LIN {X -0.057,Y -490.852,Z 943.531,A 0.000,B 0.000,C 90.000,E1 275.511} C_DIS
LIN {X 0.167,Y -491.276,Z 943.528,A 0.000,B 0.000,C 90.000,E1 274.992} C_DIS
LIN {X -0.096,Y -491.294,Z 943.525,A 0.000,B 0.000,C 90.000,E1 274.531} C_DIS
LIN {X 0.132,Y -490.916,Z 943.522,A 0.000,B 0.000,C 90.000,E1 274.012} C_DIS
LIN {X -0.165,Y -489.960,Z 943.520,A 0.000,B 0.000,C 90.000,E1 273.555} C_DIS
LIN {X 0.056,Y -488.500,Z 943.517,A 0.000,B 0.000,C 90.000,E1 273.037} C_DIS
LIN {X -0.241,Y -486.374,Z 943.514,A 0.000,B 0.000,C 90.000,E1 272.579} C_DIS
LIN {X -0.058,Y -483.567,Z 943.511,A 0.000,B 0.000,C 90.000,E1 272.064} C_DIS
LIN {X 0.120,Y -479.943,Z 943.509,A 0.000,B 0.000,C 90.000,E1 271.547} C_DIS
LIN {X -0.213,Y -475.367,Z 943.506,A 0.000,B 0.000,C 90.000,E1 271.088} C_DIS
LIN {X -0.087,Y -469.751,Z 943.503,A 0.000,B 0.000,C 90.000,E1 270.573} C_DIS
LIN {X 0.011,Y -463.745,Z 943.501,A 0.000,B 0.000,C 90.000,E1 270.115} C_DIS
LIN {X 0.069,Y -457.400,Z 943.498,A 0.000,B 0.000,C 90.000,E1 269.714} C_DIS
LIN {X 0.079,Y -450.722,Z 943.497,A 0.000,B 0.000,C 90.000,E1 269.370} C_DIS
LIN {X 0.041,Y -443.908,Z 943.495,A 0.000,B 0.000,C 90.000,E1 269.083} C_DIS
LIN {X -0.122,Y -436.692,Z 943.494,A 0.000,B 0.000,C 90.000,E1 268.854} C_DIS
LIN {X 0.080,Y -429.536,Z 943.492,A 0.000,B 0.000,C 90.000,E1 268.625} C_DIS
LIN {X 0.075,Y -421.449,Z 943.491,A 0.000,B 0.000,C 90.000,E1 268.453} C_DIS
LIN {X -0.026,Y -412.042,Z 943.491,A 0.000,B 0.000,C 90.000,E1 268.339} C_DIS
LIN {X 0.076,Y -404.135,Z 943.491,A 0.000,B 0.000,C 90.000,E1 268.282} C_DIS
LIN {X 0.000,Y -181.172,Z 943.490,A 0.000,B 0.000,C 90.000,E1 268.282} C_DIS
LIN {X -0.046,Y -180.830,Z 943.472,A 0.000,B 0.000,C 90.000,E1 264.894} C_DIS
LIN {X 0.034,Y -178.935,Z 943.443,A 0.000,B 0.000,C 90.000,E1 259.803} C_DIS
LIN {X -0.099,Y -175.985,Z 943.415,A 0.000,B 0.000,C 90.000,E1 254.755} C_DIS
LIN {X 0.016,Y -175.481,Z 943.410,A 0.000,B 0.000,C 90.000,E1 253.866} C_DIS
LIN {X 0.072,Y -172.226,Z 943.387,A 0.000,B 0.000,C 90.000,E1 249.571} C_DIS
LIN {X 0.050,Y -171.704,Z 943.382,A 0.000,B 0.000,C 90.000,E1 248.720} C_DIS
LIN {X -0.025,Y -167.298,Z 943.353,A 0.000,B 0.000,C 90.000,E1 243.563} C_DIS
LIN {X -0.019,Y -166.677,Z 943.348,A 0.000,B 0.000,C 90.000,E1 242.692} C_DIS
LIN {X -0.028,Y -162.659,Z 943.324,A 0.000,B 0.000,C 90.000,E1 238.329} C_DIS
LIN {X 0.035,Y -161.348,Z 943.314,A 0.000,B 0.000,C 90.000,E1 236.548} C_DIS
LIN {X 0.077,Y -157.342,Z 943.290,A 0.000,B 0.000,C 90.000,E1 232.110} C_DIS
LIN {X 0.009,Y -155.328,Z 943.275,A 0.000,B 0.000,C 90.000,E1 229.461} C_DIS
LIN {X -0.060,Y -151.679,Z 943.250,A 0.000,B 0.000,C 90.000,E1 225.000} C_DIS
LIN {X -0.012,Y -150.543,Z 943.240,A 0.000,B 0.000,C 90.000,E1 223.176} C_DIS
LIN {X 0.021,Y -147.269,Z 943.215,A 0.000,B 0.000,C 90.000,E1 218.624} C_DIS
LIN {X -0.006,Y -145.297,Z 943.194,A 0.000,B 0.000,C 90.000,E1 214.978} C_DIS
LIN {X -0.014,Y -142.392,Z 943.164,A 0.000,B 0.000,C 90.000,E1 209.461} C_DIS
LIN {X 0.032,Y -141.372,Z 943.148,A 0.000,B 0.000,C 90.000,E1 206.668} C_DIS
LIN {X 0.010,Y -139.346,Z 943.112,A 0.000,B 0.000,C 90.000,E1 200.174} C_DIS
LIN {X 0.015,Y -139.019,Z 943.102,A 0.000,B 0.000,C 90.000,E1 198.308} C_DIS
LIN {X 0.011,Y -138.343,Z 943.055,A 0.000,B 0.000,C 90.000,E1 189.905} C_DIS
LIN {X 0.031,Y -139.392,Z 943.008,A 0.000,B 0.000,C 90.000,E1 181.489} C_DIS
LIN {X -0.056,Y -141.291,Z 942.972,A 0.000,B 0.000,C 90.000,E1 175.008} C_DIS
LIN {X 0.043,Y -142.654,Z 942.957,A 0.000,B 0.000,C 90.000,E1 172.186} C_DIS
LIN {X -0.007,Y -144.994,Z 942.931,A 0.000,B 0.000,C 90.000,E1 167.589} C_DIS
LIN {X -0.018,Y -147.621,Z 942.911,A 0.000,B 0.000,C 90.000,E1 163.921} C_DIS
LIN {X 0.061,Y -150.247,Z 942.890,A 0.000,B 0.000,C 90.000,E1 160.242} C_DIS
LIN {X -0.066,Y -153.642,Z 942.870,A 0.000,B 0.000,C 90.000,E1 156.666} C_DIS
LIN {X -0.008,Y -157.058,Z 942.850,A 0.000,B 0.000,C 90.000,E1 153.050} C_DIS
LIN {X 0.072,Y -161.188,Z 942.830,A 0.000,B 0.000,C 90.000,E1 149.459} C_DIS
LIN {X 0.020,Y -163.281,Z 942.821,A 0.000,B 0.000,C 90.000,E1 147.709} C_DIS
LIN {X 0.031,Y -167.724,Z 942.801,A 0.000,B 0.000,C 90.000,E1 144.196} C_DIS
LIN {X -0.057,Y -171.543,Z 942.787,A 0.000,B 0.000,C 90.000,E1 141.618} C_DIS
LIN {X -0.014,Y -176.485,Z 942.768,A 0.000,B 0.000,C 90.000,E1 138.162} C_DIS
LIN {X -0.016,Y -180.782,Z 942.753,A 0.000,B 0.000,C 90.000,E1 135.607} C_DIS
LIN {X -0.028,Y -186.189,Z 942.735,A 0.000,B 0.000,C 90.000,E1 132.243} C_DIS
LIN {X 0.037,Y -190.827,Z 942.721,A 0.000,B 0.000,C 90.000,E1 129.725} C_DIS
LIN {X 0.005,Y -194.361,Z 942.709,A 0.000,B 0.000,C 90.000,E1 127.649} C_DIS
LIN {X -0.027,Y -296.822,Z 942.709,A 0.000,B 0.000,C 90.000,E1 127.649} C_DIS
LIN {X 0.038,Y -302.495,Z 942.708,A 0.000,B 0.000,C 90.000,E1 127.443} C_DIS
LIN {X 0.139,Y -304.947,Z 942.707,A 0.000,B 0.000,C 90.000,E1 127.237} C_DIS
LIN {X 0.110,Y -308.783,Z 942.705,A 0.000,B 0.000,C 90.000,E1 126.790} C_DIS
LIN {X -0.066,Y -310.657,Z 942.703,A 0.000,B 0.000,C 90.000,E1 126.503} C_DIS
LIN {X 0.007,Y -312.124,Z 942.701,A 0.000,B 0.000,C 90.000,E1 126.171} C_DIS
LIN {X 0.028,Y -314.283,Z 942.697,A 0.000,B 0.000,C 90.000,E1 125.518} C_DIS
LIN {X -0.148,Y -324.814,Z 942.680,A 0.000,B 0.000,C 90.000,E1 122.339} C_DIS
LIN {X 0.100,Y -335.642,Z 942.664,A 0.000,B 0.000,C 90.000,E1 119.461} C_DIS
LIN {X 0.012,Y -347.854,Z 942.648,A 0.000,B 0.000,C 90.000,E1 116.693} C_DIS
LIN {X 0.130,Y -361.550,Z 942.633,A 0.000,B 0.000,C 90.000,E1 113.951} C_DIS
LIN {X 0.086,Y -375.074,Z 942.620,A 0.000,B 0.000,C 90.000,E1 111.589} C_DIS
LIN {X 0.107,Y -389.967,Z 942.607,A 0.000,B 0.000,C 90.000,E1 109.268} C_DIS
LIN {X -0.132,Y -406.334,Z 942.595,A 0.000,B 0.000,C 90.000,E1 107.040} C_DIS
LIN {X -0.098,Y -424.294,Z 942.582,A 0.000,B 0.000,C 90.000,E1 104.828} C_DIS
LIN {X -0.155,Y -443.835,Z 942.570,A 0.000,B 0.000,C 90.000,E1 102.703} C_DIS
LIN {X -0.028,Y -464.124,Z 942.560,A 0.000,B 0.000,C 90.000,E1 100.715} C_DIS
LIN {X -0.116,Y -466.711,Z 942.558,A 0.000,B 0.000,C 90.000,E1 100.489} C_DIS
LIN {X -0.106,Y -468.913,Z 942.557,A 0.000,B 0.000,C 90.000,E1 100.254} C_DIS
LIN {X -0.096,Y -470.574,Z 942.556,A 0.000,B 0.000,C 90.000,E1 100.018} C_DIS
LIN {X 0.220,Y -471.940,Z 942.554,A 0.000,B 0.000,C 90.000,E1 99.726} C_DIS
LIN {X -0.007,Y -472.953,Z 942.553,A 0.000,B 0.000,C 90.000,E1 99.500} C_DIS
LIN {X 0.178,Y -474.114,Z 942.550,A 0.000,B 0.000,C 90.000,E1 98.973} C_DIS
LIN {X -0.174,Y -474.276,Z 942.547,A 0.000,B 0.000,C 90.000,E1 98.511} C_DIS
LIN {X -0.049,Y -473.471,Z 942.544,A 0.000,B 0.000,C 90.000,E1 97.992} C_DIS
LIN {X 0.079,Y -471.568,Z 942.542,A 0.000,B 0.000,C 90.000,E1 97.473} C_DIS
LIN {X -0.206,Y -468.420,Z 942.539,A 0.000,B 0.000,C 90.000,E1 97.004} C_DIS
LIN {X -0.156,Y -453.676,Z 942.526,A 0.000,B 0.000,C 90.000,E1 94.702} C_DIS
LIN {X 0.019,Y -445.560,Z 942.519,A 0.000,B 0.000,C 90.000,E1 93.383} C_DIS
LIN {X 0.147,Y -432.446,Z 942.507,A 0.000,B 0.000,C 90.000,E1 91.260} C_DIS
LIN {X -0.153,Y -415.087,Z 942.491,A 0.000,B 0.000,C 90.000,E1 88.339} C_DIS
LIN {X -0.026,Y -405.863,Z 942.482,A 0.000,B 0.000,C 90.000,E1 86.674} C_DIS
LIN {X -0.023,Y -394.990,Z 942.471,A 0.000,B 0.000,C 90.000,E1 84.723} C_DIS
LIN {X -0.178,Y -384.095,Z 942.460,A 0.000,B 0.000,C 90.000,E1 82.761} C_DIS
LIN {X -0.134,Y -374.483,Z 942.450,A 0.000,B 0.000,C 90.000,E1 81.027} C_DIS
LIN {X -0.142,Y -364.723,Z 942.440,A 0.000,B 0.000,C 90.000,E1 79.275} C_DIS
LIN {X 0.031,Y -354.702,Z 942.430,A 0.000,B 0.000,C 90.000,E1 77.465} C_DIS
LIN {X 0.005,Y -341.244,Z 942.417,A 0.000,B 0.000,C 90.000,E1 75.046} C_DIS
LIN {X -0.016,Y -325.491,Z 942.400,A 0.000,B 0.000,C 90.000,E1 71.945} C_DIS
LIN {X 0.119,Y -315.007,Z 942.387,A 0.000,B 0.000,C 90.000,E1 69.699} C_DIS
LIN {X 0.143,Y -303.085,Z 942.373,A 0.000,B 0.000,C 90.000,E1 67.102} C_DIS
LIN {X 0.120,Y -292.599,Z 942.360,A 0.000,B 0.000,C 90.000,E1 64.793} C_DIS
LIN {X 0.023,Y -283.713,Z 942.349,A 0.000,B 0.000,C 90.000,E1 62.794} C_DIS
LIN {X 0.147,Y -274.776,Z 942.337,A 0.000,B 0.000,C 90.000,E1 60.717} C_DIS
LIN {X 0.113,Y -261.660,Z 942.320,A 0.000,B 0.000,C 90.000,E1 57.582} C_DIS
LIN {X -0.077,Y -249.303,Z 942.302,A 0.000,B 0.000,C 90.000,E1 54.402} C_DIS
LIN {X -0.013,Y -238.083,Z 942.284,A 0.000,B 0.000,C 90.000,E1 51.090} C_DIS
LIN {X -0.006,Y -227.664,Z 942.265,A 0.000,B 0.000,C 90.000,E1 47.715} C_DIS
LIN {X 0.014,Y -218.081,Z 942.246,A 0.000,B 0.000,C 90.000,E1 44.271} C_DIS
LIN {X 0.049,Y -210.243,Z 942.229,A 0.000,B 0.000,C 90.000,E1 41.148} C_DIS
LIN {X -0.068,Y -202.988,Z 942.211,A 0.000,B 0.000,C 90.000,E1 38.016} C_DIS
LIN {X 0.036,Y -196.306,Z 942.193,A 0.000,B 0.000,C 90.000,E1 34.771} C_DIS
LIN {X -0.080,Y -190.148,Z 942.175,A 0.000,B 0.000,C 90.000,E1 31.544} C_DIS
LIN {X -0.059,Y -184.700,Z 942.157,A 0.000,B 0.000,C 90.000,E1 28.231} C_DIS
LIN {X 0.056,Y -179.834,Z 942.138,A 0.000,B 0.000,C 90.000,E1 24.847} C_DIS
LIN {X 0.061,Y -175.750,Z 942.119,A 0.000,B 0.000,C 90.000,E1 21.461} C_DIS
LIN {X -0.043,Y -171.472,Z 942.096,A 0.000,B 0.000,C 90.000,E1 17.221} C_DIS
LIN {X 0.026,Y -168.384,Z 942.072,A 0.000,B 0.000,C 90.000,E1 12.883} C_DIS
LIN {X 0.078,Y -165.792,Z 942.038,A 0.000,B 0.000,C 90.000,E1 6.777} C_DIS
LIN {X 0.082,Y -166.769,Z 941.968,A 0.000,B 0.000,C 90.000,E1 354.261} C_DIS
LIN {X 0.058,Y -169.679,Z 941.939,A 0.000,B 0.000,C 90.000,E1 349.050} C_DIS
LIN {X -0.015,Y -173.343,Z 941.915,A 0.000,B 0.000,C 90.000,E1 344.755} C_DIS
LIN {X -0.023,Y -177.054,Z 941.896,A 0.000,B 0.000,C 90.000,E1 341.329} C_DIS
LIN {X 0.007,Y -181.397,Z 941.877,A 0.000,B 0.000,C 90.000,E1 337.922} C_DIS
LIN {X 0.079,Y -186.476,Z 941.859,A 0.000,B 0.000,C 90.000,E1 334.537} C_DIS
LIN {X -0.067,Y -192.240,Z 941.840,A 0.000,B 0.000,C 90.000,E1 331.257} C_DIS
LIN {X 0.037,Y -198.679,Z 941.822,A 0.000,B 0.000,C 90.000,E1 327.946} C_DIS
LIN {X 0.124,Y -205.740,Z 941.804,A 0.000,B 0.000,C 90.000,E1 324.689} C_DIS
LIN {X 0.013,Y -213.322,Z 941.786,A 0.000,B 0.000,C 90.000,E1 321.537} C_DIS
LIN {X 0.031,Y -221.454,Z 941.769,A 0.000,B 0.000,C 90.000,E1 318.405} C_DIS
LIN {X 0.074,Y -230.550,Z 941.752,A 0.000,B 0.000,C 90.000,E1 315.324} C_DIS
LIN {X 0.032,Y -240.697,Z 941.735,A 0.000,B 0.000,C 90.000,E1 312.324} C_DIS
LIN {X 0.105,Y -250.556,Z 941.721,A 0.000,B 0.000,C 90.000,E1 309.725} C_DIS
LIN {X 0.034,Y -260.028,Z 941.709,A 0.000,B 0.000,C 90.000,E1 307.569} C_DIS
LIN {X -0.061,Y -272.359,Z 941.695,A 0.000,B 0.000,C 90.000,E1 305.105} C_DIS
LIN {X -0.097,Y -289.965,Z 941.678,A 0.000,B 0.000,C 90.000,E1 302.005} C_DIS
LIN {X -0.095,Y -309.009,Z 941.661,A 0.000,B 0.000,C 90.000,E1 298.999} C_DIS
LIN {X -0.154,Y -320.436,Z 941.652,A 0.000,B 0.000,C 90.000,E1 297.385} C_DIS
LIN {X 0.035,Y -335.378,Z 941.641,A 0.000,B 0.000,C 90.000,E1 295.463} C_DIS
LIN {X 0.027,Y -353.629,Z 941.630,A 0.000,B 0.000,C 90.000,E1 293.387} C_DIS
LIN {X 0.008,Y -374.769,Z 941.617,A 0.000,B 0.000,C 90.000,E1 291.153} C_DIS
LIN {X 0.065,Y -388.006,Z 941.610,A 0.000,B 0.000,C 90.000,E1 289.812} C_DIS
LIN {X 0.118,Y -400.859,Z 941.603,A 0.000,B 0.000,C 90.000,E1 288.489} C_DIS
LIN {X -0.095,Y -411.074,Z 941.597,A 0.000,B 0.000,C 90.000,E1 287.457} C_DIS
LIN {X -0.106,Y -421.008,Z 941.591,A 0.000,B 0.000,C 90.000,E1 286.386} C_DIS
LIN {X -0.109,Y -430.632,Z 941.585,A 0.000,B 0.000,C 90.000,E1 285.300} C_DIS
LIN {X -0.230,Y -439.649,Z 941.579,A 0.000,B 0.000,C 90.000,E1 284.245} C_DIS
LIN {X 0.101,Y -450.332,Z 941.572,A 0.000,B 0.000,C 90.000,E1 282.883} C_DIS
LIN {X 0.043,Y -460.450,Z 941.564,A 0.000,B 0.000,C 90.000,E1 281.591} C_DIS
LIN {X 0.197,Y -467.991,Z 941.559,A 0.000,B 0.000,C 90.000,E1 280.546} C_DIS
LIN {X -0.018,Y -474.881,Z 941.553,A 0.000,B 0.000,C 90.000,E1 279.557} C_DIS
LIN {X -0.030,Y -479.404,Z 941.549,A 0.000,B 0.000,C 90.000,E1 278.803} C_DIS
LIN {X -0.005,Y -483.183,Z 941.545,A 0.000,B 0.000,C 90.000,E1 278.049} C_DIS
LIN {X 0.171,Y -485.340,Z 941.542,A 0.000,B 0.000,C 90.000,E1 277.530} C_DIS
LIN {X -0.122,Y -487.190,Z 941.539,A 0.000,B 0.000,C 90.000,E1 277.068} C_DIS
LIN {X 0.076,Y -488.691,Z 941.536,A 0.000,B 0.000,C 90.000,E1 276.549} C_DIS
LIN {X -0.202,Y -489.902,Z 941.534,A 0.000,B 0.000,C 90.000,E1 276.087} C_DIS
LIN {X 0.015,Y -490.789,Z 941.531,A 0.000,B 0.000,C 90.000,E1 275.568} C_DIS
LIN {X 0.239,Y -491.270,Z 941.528,A 0.000,B 0.000,C 90.000,E1 275.049} C_DIS
LIN {X -0.024,Y -491.380,Z 941.525,A 0.000,B 0.000,C 90.000,E1 274.588} C_DIS
LIN {X 0.168,Y -491.060,Z 941.523,A 0.000,B 0.000,C 90.000,E1 274.073} C_DIS
LIN {X -0.094,Y -490.213,Z 941.520,A 0.000,B 0.000,C 90.000,E1 273.612} C_DIS
LIN {X 0.127,Y -488.830,Z 941.517,A 0.000,B 0.000,C 90.000,E1 273.094} C_DIS
LIN {X -0.170,Y -486.822,Z 941.515,A 0.000,B 0.000,C 90.000,E1 272.636} C_DIS
LIN {X 0.016,Y -484.126,Z 941.512,A 0.000,B 0.000,C 90.000,E1 272.121} C_DIS
LIN {X 0.196,Y -480.612,Z 941.509,A 0.000,B 0.000,C 90.000,E1 271.604} C_DIS
LIN {X 0.029,Y -478.585,Z 941.508,A 0.000,B 0.000,C 90.000,E1 271.375} C_DIS
LIN {X 0.164,Y -473.651,Z 941.505,A 0.000,B 0.000,C 90.000,E1 270.859} C_DIS
LIN {X 0.009,Y -467.978,Z 941.502,A 0.000,B 0.000,C 90.000,E1 270.401} C_DIS
LIN {X -0.217,Y -461.884,Z 941.500,A 0.000,B 0.000,C 90.000,E1 270.000} C_DIS
LIN {X -0.023,Y -455.388,Z 941.498,A 0.000,B 0.000,C 90.000,E1 269.599} C_DIS
LIN {X 0.117,Y -448.701,Z 941.496,A 0.000,B 0.000,C 90.000,E1 269.255} C_DIS
LIN {X 0.167,Y -441.816,Z 941.494,A 0.000,B 0.000,C 90.000,E1 268.969} C_DIS
LIN {X 0.114,Y -434.590,Z 941.493,A 0.000,B 0.000,C 90.000,E1 268.740} C_DIS
LIN {X -0.055,Y -427.112,Z 941.492,A 0.000,B 0.000,C 90.000,E1 268.568} C_DIS
LIN {X 0.069,Y -419.228,Z 941.491,A 0.000,B 0.000,C 90.000,E1 268.396} C_DIS
LIN {X 0.073,Y -408.844,Z 941.491,A 0.000,B 0.000,C 90.000,E1 268.282} C_DIS
LIN {X -0.088,Y -403.207,Z 941.490,A 0.000,B 0.000,C 90.000,E1 268.282} C_DIS
LIN {X -0.075,Y -181.169,Z 941.490,A 0.000,B 0.000,C 90.000,E1 268.282} C_DIS
LIN {X -0.092,Y -180.906,Z 941.474,A 0.000,B 0.000,C 90.000,E1 265.412} C_DIS
LIN {X -0.018,Y -180.696,Z 941.470,A 0.000,B 0.000,C 90.000,E1 264.546} C_DIS
LIN {X 0.060,Y -178.781,Z 941.442,A 0.000,B 0.000,C 90.000,E1 259.454} C_DIS
LIN {X -0.039,Y -175.827,Z 941.413,A 0.000,B 0.000,C 90.000,E1 254.393} C_DIS
LIN {X -0.037,Y -172.015,Z 941.385,A 0.000,B 0.000,C 90.000,E1 249.263} C_DIS
LIN {X -0.061,Y -171.437,Z 941.380,A 0.000,B 0.000,C 90.000,E1 248.411} C_DIS
LIN {X -0.007,Y -167.672,Z 941.356,A 0.000,B 0.000,C 90.000,E1 244.076} C_DIS
LIN {X -0.066,Y -166.346,Z 941.346,A 0.000,B 0.000,C 90.000,E1 242.359} C_DIS
LIN {X -0.073,Y -163.081,Z 941.327,A 0.000,B 0.000,C 90.000,E1 238.869} C_DIS
LIN {X -0.022,Y -161.023,Z 941.312,A 0.000,B 0.000,C 90.000,E1 236.215} C_DIS
LIN {X -0.037,Y -157.764,Z 941.293,A 0.000,B 0.000,C 90.000,E1 232.683} C_DIS
LIN {X 0.026,Y -155.802,Z 941.278,A 0.000,B 0.000,C 90.000,E1 229.989} C_DIS
LIN {X 0.080,Y -152.054,Z 941.253,A 0.000,B 0.000,C 90.000,E1 225.486} C_DIS
LIN {X -0.014,Y -150.304,Z 941.238,A 0.000,B 0.000,C 90.000,E1 222.813} C_DIS
LIN {X 0.023,Y -147.049,Z 941.213,A 0.000,B 0.000,C 90.000,E1 218.257} C_DIS
LIN {X 0.015,Y -145.628,Z 941.197,A 0.000,B 0.000,C 90.000,E1 215.518} C_DIS
LIN {X 0.013,Y -143.011,Z 941.172,A 0.000,B 0.000,C 90.000,E1 210.924} C_DIS
LIN {X -0.055,Y -141.638,Z 941.151,A 0.000,B 0.000,C 90.000,E1 207.257} C_DIS
LIN {X -0.005,Y -139.438,Z 941.115,A 0.000,B 0.000,C 90.000,E1 200.737} C_DIS
LIN {X 0.049,Y -139.170,Z 941.105,A 0.000,B 0.000,C 90.000,E1 198.852} C_DIS
LIN {X -0.054,Y -138.318,Z 941.053,A 0.000,B 0.000,C 90.000,E1 189.557} C_DIS
LIN {X -0.045,Y -139.473,Z 941.006,A 0.000,B 0.000,C 90.000,E1 181.146} C_DIS
LIN {X 0.035,Y -141.049,Z 940.975,A 0.000,B 0.000,C 90.000,E1 175.527} C_DIS
LIN {X -0.011,Y -142.419,Z 940.960,A 0.000,B 0.000,C 90.000,E1 172.761} C_DIS
LIN {X 0.051,Y -144.655,Z 940.934,A 0.000,B 0.000,C 90.000,E1 168.117} C_DIS
LIN {X -0.031,Y -147.852,Z 940.909,A 0.000,B 0.000,C 90.000,E1 163.559} C_DIS
LIN {X 0.053,Y -150.553,Z 940.888,A 0.000,B 0.000,C 90.000,E1 159.880} C_DIS
LIN {X -0.070,Y -154.020,Z 940.868,A 0.000,B 0.000,C 90.000,E1 156.305} C_DIS
LIN {X -0.011,Y -157.435,Z 940.848,A 0.000,B 0.000,C 90.000,E1 152.692} C_DIS
LIN {X 0.010,Y -161.650,Z 940.828,A 0.000,B 0.000,C 90.000,E1 149.125} C_DIS
LIN {X 0.028,Y -165.845,Z 940.809,A 0.000,B 0.000,C 90.000,E1 145.595} C_DIS
LIN {X 0.020,Y -170.819,Z 940.790,A 0.000,B 0.000,C 90.000,E1 142.110} C_DIS
LIN {X -0.064,Y -175.688,Z 940.770,A 0.000,B 0.000,C 90.000,E1 138.690} C_DIS
LIN {X 0.060,Y -181.301,Z 940.751,A 0.000,B 0.000,C 90.000,E1 135.243} C_DIS
LIN {X -0.068,Y -186.782,Z 940.733,A 0.000,B 0.000,C 90.000,E1 131.919} C_DIS
LIN {X 0.003,Y -191.374,Z 940.719,A 0.000,B 0.000,C 90.000,E1 129.402} C_DIS
LIN {X -0.018,Y -194.311,Z 940.709,A 0.000,B 0.000,C 90.000,E1 127.684} C_DIS
LIN {X 0.119,Y -296.535,Z 940.709,A 0.000,B 0.000,C 90.000,E1 127.649} C_DIS
LIN {X 0.077,Y -299.408,Z 940.709,A 0.000,B 0.000,C 90.000,E1 127.604} C_DIS
LIN {X -0.035,Y -304.999,Z 940.707,A 0.000,B 0.000,C 90.000,E1 127.282} C_DIS
LIN {X -0.089,Y -308.009,Z 940.705,A 0.000,B 0.000,C 90.000,E1 126.950} C_DIS
LIN {X -0.037,Y -309.993,Z 940.703,A 0.000,B 0.000,C 90.000,E1 126.629} C_DIS
LIN {X 0.081,Y -311.543,Z 940.702,A 0.000,B 0.000,C 90.000,E1 126.297} C_DIS
LIN {X -0.129,Y -312.824,Z 940.700,A 0.000,B 0.000,C 90.000,E1 126.011} C_DIS
LIN {X -0.096,Y -324.310,Z 940.680,A 0.000,B 0.000,C 90.000,E1 122.467} C_DIS
LIN {X -0.030,Y -335.074,Z 940.664,A 0.000,B 0.000,C 90.000,E1 119.617} C_DIS
LIN {X 0.030,Y -347.217,Z 940.649,A 0.000,B 0.000,C 90.000,E1 116.821} C_DIS
LIN {X 0.131,Y -360.840,Z 940.634,A 0.000,B 0.000,C 90.000,E1 114.079} C_DIS
LIN {X 0.072,Y -374.293,Z 940.621,A 0.000,B 0.000,C 90.000,E1 111.716} C_DIS
LIN {X 0.076,Y -389.110,Z 940.608,A 0.000,B 0.000,C 90.000,E1 109.396} C_DIS
LIN {X -0.061,Y -405.395,Z 940.595,A 0.000,B 0.000,C 90.000,E1 107.149} C_DIS
LIN {X -0.165,Y -423.266,Z 940.583,A 0.000,B 0.000,C 90.000,E1 104.954} C_DIS
LIN {X 0.170,Y -442.736,Z 940.571,A 0.000,B 0.000,C 90.000,E1 102.771} C_DIS
LIN {X -0.206,Y -462.995,Z 940.560,A 0.000,B 0.000,C 90.000,E1 100.838} C_DIS
LIN {X -0.188,Y -468.005,Z 940.557,A 0.000,B 0.000,C 90.000,E1 100.366} C_DIS
LIN {X -0.244,Y -469.865,Z 940.556,A 0.000,B 0.000,C 90.000,E1 100.141} C_DIS
LIN {X 0.071,Y -471.408,Z 940.555,A 0.000,B 0.000,C 90.000,E1 99.849} C_DIS
LIN {X -0.080,Y -472.562,Z 940.553,A 0.000,B 0.000,C 90.000,E1 99.613} C_DIS
LIN {X 0.026,Y -473.952,Z 940.551,A 0.000,B 0.000,C 90.000,E1 99.095} C_DIS
LIN {X 0.213,Y -474.318,Z 940.548,A 0.000,B 0.000,C 90.000,E1 98.568} C_DIS
LIN {X -0.132,Y -473.720,Z 940.545,A 0.000,B 0.000,C 90.000,E1 98.106} C_DIS
LIN {X -0.005,Y -472.069,Z 940.542,A 0.000,B 0.000,C 90.000,E1 97.587} C_DIS
LIN {X -0.146,Y -470.758,Z 940.541,A 0.000,B 0.000,C 90.000,E1 97.352} C_DIS
LIN {X -0.029,Y -456.014,Z 940.528,A 0.000,B 0.000,C 90.000,E1 95.049} C_DIS
LIN {X -0.036,Y -446.304,Z 940.519,A 0.000,B 0.000,C 90.000,E1 93.498} C_DIS
LIN {X -0.054,Y -434.857,Z 940.509,A 0.000,B 0.000,C 90.000,E1 91.661} C_DIS
LIN {X 0.150,Y -417.340,Z 940.493,A 0.000,B 0.000,C 90.000,E1 88.682} C_DIS
LIN {X -0.025,Y -406.557,Z 940.482,A 0.000,B 0.000,C 90.000,E1 86.788} C_DIS
LIN {X -0.006,Y -395.690,Z 940.471,A 0.000,B 0.000,C 90.000,E1 84.837} C_DIS
LIN {X -0.145,Y -384.775,Z 940.460,A 0.000,B 0.000,C 90.000,E1 82.875} C_DIS
LIN {X -0.087,Y -375.198,Z 940.451,A 0.000,B 0.000,C 90.000,E1 81.141} C_DIS
LIN {X -0.161,Y -363.795,Z 940.439,A 0.000,B 0.000,C 90.000,E1 79.106} C_DIS
LIN {X 0.033,Y -355.461,Z 940.431,A 0.000,B 0.000,C 90.000,E1 77.589} C_DIS
LIN {X 0.018,Y -341.999,Z 940.418,A 0.000,B 0.000,C 90.000,E1 75.172} C_DIS
LIN {X 0.149,Y -327.660,Z 940.402,A 0.000,B 0.000,C 90.000,E1 72.362} C_DIS
LIN {X -0.082,Y -317.142,Z 940.390,A 0.000,B 0.000,C 90.000,E1 70.188} C_DIS
LIN {X 0.003,Y -305.228,Z 940.375,A 0.000,B 0.000,C 90.000,E1 67.592} C_DIS
LIN {X 0.038,Y -296.244,Z 940.365,A 0.000,B 0.000,C 90.000,E1 65.613} C_DIS
LIN {X 0.119,Y -285.853,Z 940.352,A 0.000,B 0.000,C 90.000,E1 63.256} C_DIS
LIN {X -0.098,Y -276.937,Z 940.340,A 0.000,B 0.000,C 90.000,E1 61.257} C_DIS
LIN {X -0.071,Y -263.663,Z 940.323,A 0.000,B 0.000,C 90.000,E1 58.122} C_DIS
LIN {X 0.014,Y -251.132,Z 940.305,A 0.000,B 0.000,C 90.000,E1 54.895} C_DIS
LIN {X -0.027,Y -239.766,Z 940.287,A 0.000,B 0.000,C 90.000,E1 51.618} C_DIS
LIN {X 0.030,Y -229.268,Z 940.268,A 0.000,B 0.000,C 90.000,E1 48.243} C_DIS
LIN {X 0.011,Y -220.590,Z 940.251,A 0.000,B 0.000,C 90.000,E1 45.202} C_DIS
LIN {X -0.054,Y -212.608,Z 940.234,A 0.000,B 0.000,C 90.000,E1 42.123} C_DIS
LIN {X 0.018,Y -205.261,Z 940.216,A 0.000,B 0.000,C 90.000,E1 38.955} C_DIS
LIN {X 0.011,Y -198.392,Z 940.199,A 0.000,B 0.000,C 90.000,E1 35.758} C_DIS
LIN {X -0.108,Y -192.106,Z 940.181,A 0.000,B 0.000,C 90.000,E1 32.546} C_DIS
LIN {X 0.054,Y -186.458,Z 940.162,A 0.000,B 0.000,C 90.000,E1 29.205} C_DIS
LIN {X -0.038,Y -181.394,Z 940.144,A 0.000,B 0.000,C 90.000,E1 25.899} C_DIS
LIN {X 0.002,Y -177.092,Z 940.125,A 0.000,B 0.000,C 90.000,E1 22.514} C_DIS
LIN {X 0.053,Y -172.600,Z 940.101,A 0.000,B 0.000,C 90.000,E1 18.236} C_DIS
LIN {X 0.031,Y -169.240,Z 940.078,A 0.000,B 0.000,C 90.000,E1 13.939} C_DIS
LIN {X -0.008,Y -166.604,Z 940.049,A 0.000,B 0.000,C 90.000,E1 8.746} C_DIS
LIN {X -0.044,Y -166.673,Z 939.973,A 0.000,B 0.000,C 90.000,E1 355.179} C_DIS
LIN {X 0.050,Y -169.353,Z 939.944,A 0.000,B 0.000,C 90.000,E1 349.926} C_DIS
LIN {X -0.076,Y -172.783,Z 939.920,A 0.000,B 0.000,C 90.000,E1 345.644} C_DIS
LIN {X 0.017,Y -176.324,Z 939.901,A 0.000,B 0.000,C 90.000,E1 342.181} C_DIS
LIN {X 0.031,Y -180.513,Z 939.882,A 0.000,B 0.000,C 90.000,E1 338.773} C_DIS
LIN {X 0.011,Y -185.381,Z 939.863,A 0.000,B 0.000,C 90.000,E1 335.409} C_DIS
LIN {X -0.075,Y -190.977,Z 939.845,A 0.000,B 0.000,C 90.000,E1 332.103} C_DIS
LIN {X 0.000,Y -197.271,Z 939.827,A 0.000,B 0.000,C 90.000,E1 328.791} C_DIS
LIN {X -0.002,Y -204.162,Z 939.809,A 0.000,B 0.000,C 90.000,E1 325.548} C_DIS
LIN {X 0.006,Y -211.659,Z 939.791,A 0.000,B 0.000,C 90.000,E1 322.351} C_DIS
LIN {X -0.026,Y -219.601,Z 939.773,A 0.000,B 0.000,C 90.000,E1 319.218} C_DIS
LIN {X -0.020,Y -228.434,Z 939.756,A 0.000,B 0.000,C 90.000,E1 316.134} C_DIS
LIN {X 0.041,Y -238.287,Z 939.739,A 0.000,B 0.000,C 90.000,E1 313.095} C_DIS
LIN {X -0.131,Y -249.288,Z 939.723,A 0.000,B 0.000,C 90.000,E1 310.172} C_DIS
LIN {X -0.031,Y -258.583,Z 939.711,A 0.000,B 0.000,C 90.000,E1 307.971} C_DIS
LIN {X 0.097,Y -268.834,Z 939.699,A 0.000,B 0.000,C 90.000,E1 305.804} C_DIS
LIN {X 0.006,Y -283.998,Z 939.684,A 0.000,B 0.000,C 90.000,E1 303.038} C_DIS
LIN {X 0.007,Y -302.413,Z 939.667,A 0.000,B 0.000,C 90.000,E1 300.001} C_DIS
LIN {X -0.054,Y -317.966,Z 939.654,A 0.000,B 0.000,C 90.000,E1 297.719} C_DIS
LIN {X -0.012,Y -332.758,Z 939.643,A 0.000,B 0.000,C 90.000,E1 295.796} C_DIS
LIN {X -0.060,Y -353.678,Z 939.630,A 0.000,B 0.000,C 90.000,E1 293.387} C_DIS
LIN {X -0.024,Y -372.218,Z 939.619,A 0.000,B 0.000,C 90.000,E1 291.408} C_DIS
LIN {X -0.072,Y -388.032,Z 939.610,A 0.000,B 0.000,C 90.000,E1 289.812} C_DIS
LIN {X -0.089,Y -400.921,Z 939.603,A 0.000,B 0.000,C 90.000,E1 288.489} C_DIS
LIN {X 0.147,Y -411.080,Z 939.597,A 0.000,B 0.000,C 90.000,E1 287.402} C_DIS
LIN {X 0.246,Y -420.999,Z 939.591,A 0.000,B 0.000,C 90.000,E1 286.315} C_DIS
LIN {X 0.139,Y -430.654,Z 939.585,A 0.000,B 0.000,C 90.000,E1 285.245} C_DIS
LIN {X -0.089,Y -441.831,Z 939.577,A 0.000,B 0.000,C 90.000,E1 283.939} C_DIS
LIN {X 0.166,Y -452.442,Z 939.570,A 0.000,B 0.000,C 90.000,E1 282.591} C_DIS
LIN {X -0.134,Y -460.506,Z 939.564,A 0.000,B 0.000,C 90.000,E1 281.591} C_DIS
LIN {X 0.017,Y -468.015,Z 939.559,A 0.000,B 0.000,C 90.000,E1 280.546} C_DIS
LIN {X -0.200,Y -474.931,Z 939.553,A 0.000,B 0.000,C 90.000,E1 279.557} C_DIS
LIN {X -0.213,Y -479.427,Z 939.549,A 0.000,B 0.000,C 90.000,E1 278.803} C_DIS
LIN {X -0.189,Y -483.221,Z 939.545,A 0.000,B 0.000,C 90.000,E1 278.049} C_DIS
LIN {X -0.014,Y -485.375,Z 939.542,A 0.000,B 0.000,C 90.000,E1 277.530} C_DIS
LIN {X 0.176,Y -487.229,Z 939.539,A 0.000,B 0.000,C 90.000,E1 277.011} C_DIS
LIN {X -0.054,Y -488.742,Z 939.536,A 0.000,B 0.000,C 90.000,E1 276.543} C_DIS
LIN {X 0.099,Y -489.960,Z 939.534,A 0.000,B 0.000,C 90.000,E1 276.030} C_DIS
LIN {X -0.171,Y -490.812,Z 939.531,A 0.000,B 0.000,C 90.000,E1 275.568} C_DIS
LIN {X 0.052,Y -491.326,Z 939.528,A 0.000,B 0.000,C 90.000,E1 275.049} C_DIS
LIN {X -0.211,Y -491.439,Z 939.525,A 0.000,B 0.000,C 90.000,E1 274.588} C_DIS
LIN {X -0.019,Y -491.075,Z 939.523,A 0.000,B 0.000,C 90.000,E1 274.073} C_DIS
LIN {X 0.210,Y -490.225,Z 939.520,A 0.000,B 0.000,C 90.000,E1 273.555} C_DIS
LIN {X -0.057,Y -488.846,Z 939.517,A 0.000,B 0.000,C 90.000,E1 273.094} C_DIS
LIN {X 0.133,Y -486.841,Z 939.514,A 0.000,B 0.000,C 90.000,E1 272.579} C_DIS
LIN {X -0.167,Y -484.121,Z 939.512,A 0.000,B 0.000,C 90.000,E1 272.121} C_DIS
LIN {X 0.158,Y -482.504,Z 939.510,A 0.000,B 0.000,C 90.000,E1 271.835} C_DIS
LIN {X -0.151,Y -478.558,Z 939.508,A 0.000,B 0.000,C 90.000,E1 271.375} C_DIS
LIN {X -0.015,Y -473.637,Z 939.505,A 0.000,B 0.000,C 90.000,E1 270.859} C_DIS
LIN {X -0.168,Y -467.966,Z 939.502,A 0.000,B 0.000,C 90.000,E1 270.401} C_DIS
LIN {X 0.096,Y -461.876,Z 939.500,A 0.000,B 0.000,C 90.000,E1 269.943} C_DIS
LIN {X -0.139,Y -455.456,Z 939.498,A 0.000,B 0.000,C 90.000,E1 269.599} C_DIS
LIN {X 0.028,Y -448.865,Z 939.496,A 0.000,B 0.000,C 90.000,E1 269.255} C_DIS
LIN {X 0.098,Y -442.072,Z 939.494,A 0.000,B 0.000,C 90.000,E1 268.969} C_DIS
LIN {X 0.041,Y -434.928,Z 939.493,A 0.000,B 0.000,C 90.000,E1 268.740} C_DIS
LIN {X -0.135,Y -427.516,Z 939.492,A 0.000,B 0.000,C 90.000,E1 268.568} C_DIS
LIN {X -0.020,Y -419.686,Z 939.491,A 0.000,B 0.000,C 90.000,E1 268.396} C_DIS
LIN {X -0.025,Y -409.718,Z 939.490,A 0.000,B 0.000,C 90.000,E1 268.282} C_DIS
LIN {X 0.175,Y -404.707,Z 939.490,A 0.000,B 0.000,C 90.000,E1 268.224} C_DIS
LIN {X 0.060,Y -181.166,Z 939.490,A 0.000,B 0.000,C 90.000,E1 268.224} C_DIS
LIN {X 0.042,Y -180.906,Z 939.474,A 0.000,B 0.000,C 90.000,E1 265.355} C_DIS
LIN {X -0.064,Y -180.688,Z 939.470,A 0.000,B 0.000,C 90.000,E1 264.546} C_DIS
LIN {X 0.014,Y -178.772,Z 939.441,A 0.000,B 0.000,C 90.000,E1 259.454} C_DIS
LIN {X -0.083,Y -175.819,Z 939.413,A 0.000,B 0.000,C 90.000,E1 254.393} C_DIS
LIN {X 0.080,Y -172.006,Z 939.385,A 0.000,B 0.000,C 90.000,E1 249.209} C_DIS
LIN {X 0.054,Y -171.423,Z 939.380,A 0.000,B 0.000,C 90.000,E1 248.358} C_DIS
LIN {X -0.050,Y -167.661,Z 939.356,A 0.000,B 0.000,C 90.000,E1 244.076} C_DIS
LIN {X 0.038,Y -166.330,Z 939.346,A 0.000,B 0.000,C 90.000,E1 242.308} C_DIS
LIN {X 0.023,Y -163.069,Z 939.327,A 0.000,B 0.000,C 90.000,E1 238.820} C_DIS
LIN {X -0.064,Y -161.008,Z 939.312,A 0.000,B 0.000,C 90.000,E1 236.215} C_DIS
LIN {X 0.046,Y -157.752,Z 939.293,A 0.000,B 0.000,C 90.000,E1 232.637} C_DIS
LIN {X -0.016,Y -155.790,Z 939.278,A 0.000,B 0.000,C 90.000,E1 229.989} C_DIS
LIN {X 0.038,Y -152.043,Z 939.253,A 0.000,B 0.000,C 90.000,E1 225.486} C_DIS
LIN {X 0.056,Y -150.293,Z 939.238,A 0.000,B 0.000,C 90.000,E1 222.771} C_DIS
LIN {X -0.018,Y -147.040,Z 939.213,A 0.000,B 0.000,C 90.000,E1 218.257} C_DIS
LIN {X -0.025,Y -145.620,Z 939.197,A 0.000,B 0.000,C 90.000,E1 215.518} C_DIS
LIN {X -0.027,Y -143.004,Z 939.172,A 0.000,B 0.000,C 90.000,E1 210.924} C_DIS
LIN {X 0.031,Y -141.631,Z 939.151,A 0.000,B 0.000,C 90.000,E1 207.206} C_DIS
LIN {X -0.044,Y -139.435,Z 939.115,A 0.000,B 0.000,C 90.000,E1 200.737} C_DIS
LIN {X 0.010,Y -139.166,Z 939.105,A 0.000,B 0.000,C 90.000,E1 198.852} C_DIS
LIN {X 0.044,Y -138.316,Z 939.053,A 0.000,B 0.000,C 90.000,E1 189.500} C_DIS
LIN {X 0.055,Y -139.475,Z 939.006,A 0.000,B 0.000,C 90.000,E1 181.088} C_DIS
LIN {X -0.004,Y -141.056,Z 938.975,A 0.000,B 0.000,C 90.000,E1 175.527} C_DIS
LIN {X -0.050,Y -142.427,Z 938.960,A 0.000,B 0.000,C 90.000,E1 172.761} C_DIS
LIN {X 0.011,Y -144.665,Z 938.934,A 0.000,B 0.000,C 90.000,E1 168.117} C_DIS
LIN {X -0.005,Y -147.249,Z 938.914,A 0.000,B 0.000,C 90.000,E1 164.448} C_DIS
LIN {X 0.012,Y -150.566,Z 938.888,A 0.000,B 0.000,C 90.000,E1 159.880} C_DIS
LIN {X 0.091,Y -154.035,Z 938.868,A 0.000,B 0.000,C 90.000,E1 156.230} C_DIS
LIN {X 0.019,Y -157.451,Z 938.848,A 0.000,B 0.000,C 90.000,E1 152.666} C_DIS
LIN {X -0.033,Y -161.669,Z 938.828,A 0.000,B 0.000,C 90.000,E1 149.125} C_DIS
LIN {X -0.015,Y -165.865,Z 938.809,A 0.000,B 0.000,C 90.000,E1 145.595} C_DIS
LIN {X -0.024,Y -170.842,Z 938.789,A 0.000,B 0.000,C 90.000,E1 142.110} C_DIS
LIN {X 0.024,Y -175.711,Z 938.770,A 0.000,B 0.000,C 90.000,E1 138.647} C_DIS
LIN {X 0.014,Y -181.322,Z 938.751,A 0.000,B 0.000,C 90.000,E1 135.243} C_DIS
LIN {X 0.010,Y -186.807,Z 938.733,A 0.000,B 0.000,C 90.000,E1 131.881} C_DIS
LIN {X -0.045,Y -191.398,Z 938.719,A 0.000,B 0.000,C 90.000,E1 129.402} C_DIS
LIN {X -0.091,Y -194.269,Z 938.709,A 0.000,B 0.000,C 90.000,E1 127.729} C_DIS
LIN {X 0.042,Y -297.301,Z 938.709,A 0.000,B 0.000,C 90.000,E1 127.684} C_DIS
LIN {X 0.117,Y -298.411,Z 938.709,A 0.000,B 0.000,C 90.000,E1 127.649} C_DIS
LIN {X -0.026,Y -302.625,Z 938.708,A 0.000,B 0.000,C 90.000,E1 127.488} C_DIS
LIN {X 0.069,Y -304.984,Z 938.707,A 0.000,B 0.000,C 90.000,E1 127.282} C_DIS
LIN {X -0.165,Y -308.205,Z 938.705,A 0.000,B 0.000,C 90.000,E1 126.950} C_DIS
LIN {X 0.104,Y -310.152,Z 938.703,A 0.000,B 0.000,C 90.000,E1 126.583} C_DIS
LIN {X -0.060,Y -311.672,Z 938.702,A 0.000,B 0.000,C 90.000,E1 126.297} C_DIS
LIN {X -0.018,Y -312.903,Z 938.700,A 0.000,B 0.000,C 90.000,E1 125.964} C_DIS
LIN {X 0.033,Y -324.379,Z 938.680,A 0.000,B 0.000,C 90.000,E1 122.418} C_DIS
LIN {X -0.011,Y -335.154,Z 938.664,A 0.000,B 0.000,C 90.000,E1 119.589} C_DIS
LIN {X 0.038,Y -347.310,Z 938.649,A 0.000,B 0.000,C 90.000,E1 116.796} C_DIS
LIN {X -0.022,Y -360.946,Z 938.634,A 0.000,B 0.000,C 90.000,E1 114.079} C_DIS
LIN {X -0.084,Y -374.413,Z 938.621,A 0.000,B 0.000,C 90.000,E1 111.716} C_DIS
LIN {X -0.084,Y -389.243,Z 938.608,A 0.000,B 0.000,C 90.000,E1 109.396} C_DIS
LIN {X 0.165,Y -405.543,Z 938.595,A 0.000,B 0.000,C 90.000,E1 107.094} C_DIS
LIN {X 0.079,Y -423.431,Z 938.583,A 0.000,B 0.000,C 90.000,E1 104.898} C_DIS
LIN {X 0.005,Y -442.915,Z 938.571,A 0.000,B 0.000,C 90.000,E1 102.771} C_DIS
LIN {X 0.089,Y -463.179,Z 938.560,A 0.000,B 0.000,C 90.000,E1 100.782} C_DIS
LIN {X 0.113,Y -468.155,Z 938.557,A 0.000,B 0.000,C 90.000,E1 100.310} C_DIS
LIN {X 0.144,Y -469.977,Z 938.556,A 0.000,B 0.000,C 90.000,E1 100.074} C_DIS
LIN {X -0.087,Y -471.489,Z 938.555,A 0.000,B 0.000,C 90.000,E1 99.849} C_DIS
LIN {X 0.230,Y -472.620,Z 938.553,A 0.000,B 0.000,C 90.000,E1 99.557} C_DIS
LIN {X -0.131,Y -473.973,Z 938.550,A 0.000,B 0.000,C 90.000,E1 99.095} C_DIS
LIN {X 0.057,Y -474.305,Z 938.548,A 0.000,B 0.000,C 90.000,E1 98.568} C_DIS
LIN {X 0.180,Y -473.676,Z 938.545,A 0.000,B 0.000,C 90.000,E1 98.049} C_DIS
LIN {X -0.161,Y -471.985,Z 938.542,A 0.000,B 0.000,C 90.000,E1 97.587} C_DIS
LIN {X 0.165,Y -470.649,Z 938.541,A 0.000,B 0.000,C 90.000,E1 97.296} C_DIS
LIN {X -0.183,Y -455.949,Z 938.528,A 0.000,B 0.000,C 90.000,E1 95.049} C_DIS
LIN {X -0.187,Y -446.265,Z 938.519,A 0.000,B 0.000,C 90.000,E1 93.498} C_DIS
LIN {X -0.201,Y -434.844,Z 938.509,A 0.000,B 0.000,C 90.000,E1 91.661} C_DIS
LIN {X 0.007,Y -417.290,Z 938.493,A 0.000,B 0.000,C 90.000,E1 88.682} C_DIS
LIN {X -0.165,Y -406.509,Z 938.482,A 0.000,B 0.000,C 90.000,E1 86.788} C_DIS
LIN {X -0.144,Y -395.623,Z 938.471,A 0.000,B 0.000,C 90.000,E1 84.837} C_DIS
LIN {X 0.102,Y -384.694,Z 938.460,A 0.000,B 0.000,C 90.000,E1 82.818} C_DIS
LIN {X 0.163,Y -373.489,Z 938.449,A 0.000,B 0.000,C 90.000,E1 80.792} C_DIS
LIN {X 0.065,Y -363.697,Z 938.439,A 0.000,B 0.000,C 90.000,E1 79.050} C_DIS
LIN {X -0.096,Y -355.370,Z 938.431,A 0.000,B 0.000,C 90.000,E1 77.589} C_DIS
LIN {X -0.108,Y -341.924,Z 938.418,A 0.000,B 0.000,C 90.000,E1 75.172} C_DIS
LIN {X 0.026,Y -327.583,Z 938.402,A 0.000,B 0.000,C 90.000,E1 72.362} C_DIS
LIN {X 0.095,Y -317.079,Z 938.390,A 0.000,B 0.000,C 90.000,E1 70.134} C_DIS
LIN {X 0.168,Y -305.179,Z 938.375,A 0.000,B 0.000,C 90.000,E1 67.539} C_DIS
LIN {X -0.076,Y -296.195,Z 938.364,A 0.000,B 0.000,C 90.000,E1 65.613} C_DIS
LIN {X -0.020,Y -284.314,Z 938.350,A 0.000,B 0.000,C 90.000,E1 62.922} C_DIS
LIN {X -0.017,Y -275.354,Z 938.338,A 0.000,B 0.000,C 90.000,E1 60.873} C_DIS
LIN {X -0.037,Y -262.122,Z 938.321,A 0.000,B 0.000,C 90.000,E1 57.740} C_DIS
LIN {X 0.132,Y -249.708,Z 938.303,A 0.000,B 0.000,C 90.000,E1 54.482} C_DIS
LIN {X -0.140,Y -238.483,Z 938.285,A 0.000,B 0.000,C 90.000,E1 51.251} C_DIS
LIN {X 0.034,Y -228.097,Z 938.266,A 0.000,B 0.000,C 90.000,E1 47.838} C_DIS
LIN {X -0.083,Y -218.534,Z 938.247,A 0.000,B 0.000,C 90.000,E1 44.433} C_DIS
LIN {X -0.032,Y -210.767,Z 938.229,A 0.000,B 0.000,C 90.000,E1 41.310} C_DIS
LIN {X -0.005,Y -203.566,Z 938.212,A 0.000,B 0.000,C 90.000,E1 38.141} C_DIS
LIN {X -0.056,Y -196.878,Z 938.194,A 0.000,B 0.000,C 90.000,E1 34.945} C_DIS
LIN {X -0.001,Y -190.732,Z 938.176,A 0.000,B 0.000,C 90.000,E1 31.671} C_DIS
LIN {X 0.031,Y -185.277,Z 938.158,A 0.000,B 0.000,C 90.000,E1 28.359} C_DIS
LIN {X -0.006,Y -180.396,Z 938.139,A 0.000,B 0.000,C 90.000,E1 25.027} C_DIS
LIN {X -0.053,Y -176.294,Z 938.120,A 0.000,B 0.000,C 90.000,E1 21.663} C_DIS
LIN {X -0.075,Y -172.005,Z 938.097,A 0.000,B 0.000,C 90.000,E1 17.402} C_DIS
LIN {X 0.012,Y -168.880,Z 938.073,A 0.000,B 0.000,C 90.000,E1 13.063} C_DIS
LIN {X -0.040,Y -166.505,Z 938.044,A 0.000,B 0.000,C 90.000,E1 7.871} C_DIS
LIN {X -0.068,Y -167.266,Z 937.968,A 0.000,B 0.000,C 90.000,E1 354.318} C_DIS
LIN {X 0.066,Y -169.613,Z 937.944,A 0.000,B 0.000,C 90.000,E1 349.926} C_DIS
LIN {X -0.051,Y -173.050,Z 937.920,A 0.000,B 0.000,C 90.000,E1 345.644} C_DIS
LIN {X 0.043,Y -177.571,Z 937.896,A 0.000,B 0.000,C 90.000,E1 341.329} C_DIS
LIN {X -0.080,Y -181.910,Z 937.878,A 0.000,B 0.000,C 90.000,E1 337.975} C_DIS
LIN {X 0.007,Y -186.959,Z 937.859,A 0.000,B 0.000,C 90.000,E1 334.588} C_DIS
LIN {X 0.045,Y -192.705,Z 937.840,A 0.000,B 0.000,C 90.000,E1 331.257} C_DIS
LIN {X -0.005,Y -199.219,Z 937.822,A 0.000,B 0.000,C 90.000,E1 327.995} C_DIS
LIN {X -0.018,Y -206.229,Z 937.804,A 0.000,B 0.000,C 90.000,E1 324.769} C_DIS
LIN {X -0.125,Y -213.845,Z 937.787,A 0.000,B 0.000,C 90.000,E1 321.618} C_DIS
LIN {X 0.047,Y -221.958,Z 937.769,A 0.000,B 0.000,C 90.000,E1 318.447} C_DIS
LIN {X -0.049,Y -231.042,Z 937.752,A 0.000,B 0.000,C 90.000,E1 315.405} C_DIS
LIN {X 0.079,Y -241.179,Z 937.735,A 0.000,B 0.000,C 90.000,E1 312.366} C_DIS
LIN {X -0.003,Y -250.976,Z 937.721,A 0.000,B 0.000,C 90.000,E1 309.806} C_DIS
LIN {X -0.032,Y -262.042,Z 937.707,A 0.000,B 0.000,C 90.000,E1 307.282} C_DIS
LIN {X -0.079,Y -274.425,Z 937.693,A 0.000,B 0.000,C 90.000,E1 304.818} C_DIS
LIN {X -0.067,Y -291.987,Z 937.676,A 0.000,B 0.000,C 90.000,E1 301.720} C_DIS
LIN {X 0.118,Y -311.047,Z 937.660,A 0.000,B 0.000,C 90.000,E1 298.693} C_DIS
LIN {X 0.097,Y -322.603,Z 937.651,A 0.000,B 0.000,C 90.000,E1 297.078} C_DIS
LIN {X -0.001,Y -337.681,Z 937.640,A 0.000,B 0.000,C 90.000,E1 295.207} C_DIS
LIN {X 0.048,Y -361.506,Z 937.625,A 0.000,B 0.000,C 90.000,E1 292.514} C_DIS
LIN {X 0.131,Y -380.213,Z 937.614,A 0.000,B 0.000,C 90.000,E1 290.556} C_DIS
LIN {X -0.052,Y -393.149,Z 937.607,A 0.000,B 0.000,C 90.000,E1 289.268} C_DIS
LIN {X -0.099,Y -405.993,Z 937.600,A 0.000,B 0.000,C 90.000,E1 287.946} C_DIS
LIN {X -0.003,Y -416.157,Z 937.594,A 0.000,B 0.000,C 90.000,E1 286.858} C_DIS
LIN {X -0.118,Y -425.994,Z 937.588,A 0.000,B 0.000,C 90.000,E1 285.788} C_DIS
LIN {X 0.067,Y -433.043,Z 937.583,A 0.000,B 0.000,C 90.000,E1 284.954} C_DIS
LIN {X -0.133,Y -444.073,Z 937.576,A 0.000,B 0.000,C 90.000,E1 283.647} C_DIS
LIN {X 0.164,Y -454.606,Z 937.568,A 0.000,B 0.000,C 90.000,E1 282.299} C_DIS
LIN {X -0.113,Y -462.533,Z 937.563,A 0.000,B 0.000,C 90.000,E1 281.299} C_DIS
LIN {X 0.064,Y -469.896,Z 937.557,A 0.000,B 0.000,C 90.000,E1 280.254} C_DIS
LIN {X 0.005,Y -475.032,Z 937.553,A 0.000,B 0.000,C 90.000,E1 279.500} C_DIS
LIN {X -0.004,Y -479.526,Z 937.549,A 0.000,B 0.000,C 90.000,E1 278.746} C_DIS
LIN {X 0.023,Y -483.298,Z 937.544,A 0.000,B 0.000,C 90.000,E1 277.992} C_DIS
LIN {X 0.200,Y -485.431,Z 937.542,A 0.000,B 0.000,C 90.000,E1 277.473} C_DIS
LIN {X -0.032,Y -487.305,Z 937.539,A 0.000,B 0.000,C 90.000,E1 277.004} C_DIS
LIN {X 0.163,Y -488.824,Z 937.536,A 0.000,B 0.000,C 90.000,E1 276.486} C_DIS
LIN {X -0.117,Y -490.006,Z 937.533,A 0.000,B 0.000,C 90.000,E1 276.024} C_DIS
LIN {X 0.049,Y -490.896,Z 937.531,A 0.000,B 0.000,C 90.000,E1 275.511} C_DIS
LIN {X -0.215,Y -491.380,Z 937.528,A 0.000,B 0.000,C 90.000,E1 275.049} C_DIS
LIN {X 0.012,Y -491.471,Z 937.525,A 0.000,B 0.000,C 90.000,E1 274.531} C_DIS
LIN {X 0.239,Y -491.115,Z 937.522,A 0.000,B 0.000,C 90.000,E1 274.012} C_DIS
LIN {X -0.056,Y -490.275,Z 937.520,A 0.000,B 0.000,C 90.000,E1 273.555} C_DIS
LIN {X 0.165,Y -488.860,Z 937.517,A 0.000,B 0.000,C 90.000,E1 273.037} C_DIS
LIN {X -0.131,Y -486.847,Z 937.514,A 0.000,B 0.000,C 90.000,E1 272.579} C_DIS
LIN {X 0.054,Y -484.103,Z 937.511,A 0.000,B 0.000,C 90.000,E1 272.064} C_DIS
LIN {X 0.234,Y -480.550,Z 937.509,A 0.000,B 0.000,C 90.000,E1 271.547} C_DIS
LIN {X 0.068,Y -478.494,Z 937.507,A 0.000,B 0.000,C 90.000,E1 271.318} C_DIS
LIN {X 0.202,Y -473.503,Z 937.505,A 0.000,B 0.000,C 90.000,E1 270.802} C_DIS
LIN {X 0.047,Y -467.810,Z 937.502,A 0.000,B 0.000,C 90.000,E1 270.344} C_DIS
LIN {X -0.161,Y -461.691,Z 937.500,A 0.000,B 0.000,C 90.000,E1 269.943} C_DIS
LIN {X 0.087,Y -455.238,Z 937.497,A 0.000,B 0.000,C 90.000,E1 269.542} C_DIS
LIN {X -0.181,Y -448.652,Z 937.496,A 0.000,B 0.000,C 90.000,E1 269.255} C_DIS
LIN {X -0.132,Y -441.744,Z 937.494,A 0.000,B 0.000,C 90.000,E1 268.969} C_DIS
LIN {X -0.187,Y -434.576,Z 937.493,A 0.000,B 0.000,C 90.000,E1 268.740} C_DIS
LIN {X 0.081,Y -427.228,Z 937.492,A 0.000,B 0.000,C 90.000,E1 268.511} C_DIS
LIN {X -0.205,Y -419.429,Z 937.491,A 0.000,B 0.000,C 90.000,E1 268.396} C_DIS
LIN {X -0.182,Y -409.849,Z 937.490,A 0.000,B 0.000,C 90.000,E1 268.282} C_DIS
LIN {X 0.064,Y -406.397,Z 937.490,A 0.000,B 0.000,C 90.000,E1 268.224} C_DIS
LIN {X -0.008,Y -181.162,Z 937.490,A 0.000,B 0.000,C 90.000,E1 268.224} C_DIS
LIN {X -0.024,Y -180.906,Z 937.474,A 0.000,B 0.000,C 90.000,E1 265.355} C_DIS
LIN {X 0.049,Y -180.677,Z 937.469,A 0.000,B 0.000,C 90.000,E1 264.489} C_DIS
LIN {X -0.052,Y -178.760,Z 937.441,A 0.000,B 0.000,C 90.000,E1 259.454} C_DIS
LIN {X 0.020,Y -175.807,Z 937.413,A 0.000,B 0.000,C 90.000,E1 254.338} C_DIS
LIN {X 0.015,Y -171.992,Z 937.385,A 0.000,B 0.000,C 90.000,E1 249.209} C_DIS
LIN {X 0.053,Y -171.404,Z 937.380,A 0.000,B 0.000,C 90.000,E1 248.337} C_DIS
LIN {X 0.037,Y -167.645,Z 937.356,A 0.000,B 0.000,C 90.000,E1 244.024} C_DIS
LIN {X 0.052,Y -166.308,Z 937.346,A 0.000,B 0.000,C 90.000,E1 242.281} C_DIS
LIN {X 0.045,Y -163.050,Z 937.327,A 0.000,B 0.000,C 90.000,E1 238.791} C_DIS
LIN {X 0.007,Y -160.984,Z 937.312,A 0.000,B 0.000,C 90.000,E1 236.167} C_DIS
LIN {X -0.016,Y -157.734,Z 937.292,A 0.000,B 0.000,C 90.000,E1 232.637} C_DIS
LIN {X -0.077,Y -155.773,Z 937.278,A 0.000,B 0.000,C 90.000,E1 229.989} C_DIS
LIN {X -0.022,Y -152.028,Z 937.253,A 0.000,B 0.000,C 90.000,E1 225.486} C_DIS
LIN {X -0.004,Y -150.276,Z 937.238,A 0.000,B 0.000,C 90.000,E1 222.771} C_DIS
LIN {X 0.014,Y -147.027,Z 937.212,A 0.000,B 0.000,C 90.000,E1 218.222} C_DIS
LIN {X 0.035,Y -145.608,Z 937.197,A 0.000,B 0.000,C 90.000,E1 215.471} C_DIS
LIN {X 0.038,Y -142.994,Z 937.172,A 0.000,B 0.000,C 90.000,E1 210.875} C_DIS
LIN {X -0.026,Y -141.621,Z 937.151,A 0.000,B 0.000,C 90.000,E1 207.206} C_DIS
LIN {X 0.030,Y -139.432,Z 937.115,A 0.000,B 0.000,C 90.000,E1 200.684} C_DIS
LIN {X -0.047,Y -139.162,Z 937.105,A 0.000,B 0.000,C 90.000,E1 198.852} C_DIS
LIN {X -0.010,Y -138.341,Z 937.058,A 0.000,B 0.000,C 90.000,E1 190.433} C_DIS
LIN {X -0.002,Y -139.479,Z 937.006,A 0.000,B 0.000,C 90.000,E1 181.088} C_DIS
LIN {X -0.062,Y -141.066,Z 936.975,A 0.000,B 0.000,C 90.000,E1 175.527} C_DIS
LIN {X 0.033,Y -142.440,Z 936.960,A 0.000,B 0.000,C 90.000,E1 172.704} C_DIS
LIN {X -0.047,Y -144.678,Z 936.934,A 0.000,B 0.000,C 90.000,E1 168.117} C_DIS
LIN {X 0.077,Y -147.268,Z 936.913,A 0.000,B 0.000,C 90.000,E1 164.393} C_DIS
LIN {X -0.048,Y -150.585,Z 936.888,A 0.000,B 0.000,C 90.000,E1 159.880} C_DIS
LIN {X 0.031,Y -154.057,Z 936.868,A 0.000,B 0.000,C 90.000,E1 156.230} C_DIS
LIN {X -0.042,Y -157.476,Z 936.848,A 0.000,B 0.000,C 90.000,E1 152.666} C_DIS
LIN {X 0.043,Y -161.699,Z 936.828,A 0.000,B 0.000,C 90.000,E1 149.076} C_DIS
LIN {X -0.079,Y -165.893,Z 936.809,A 0.000,B 0.000,C 90.000,E1 145.595} C_DIS
LIN {X 0.046,Y -170.876,Z 936.789,A 0.000,B 0.000,C 90.000,E1 142.065} C_DIS
LIN {X 0.074,Y -175.744,Z 936.770,A 0.000,B 0.000,C 90.000,E1 138.609} C_DIS
LIN {X -0.053,Y -181.354,Z 936.751,A 0.000,B 0.000,C 90.000,E1 135.243} C_DIS
LIN {X 0.080,Y -186.845,Z 936.733,A 0.000,B 0.000,C 90.000,E1 131.838} C_DIS
LIN {X 0.034,Y -191.431,Z 936.719,A 0.000,B 0.000,C 90.000,E1 129.358} C_DIS
LIN {X 0.025,Y -194.208,Z 936.710,A 0.000,B 0.000,C 90.000,E1 127.729} C_DIS
LIN {X -0.007,Y -296.496,Z 936.710,A 0.000,B 0.000,C 90.000,E1 127.729} C_DIS
LIN {X 0.114,Y -300.487,Z 936.709,A 0.000,B 0.000,C 90.000,E1 127.604} C_DIS
LIN {X -0.033,Y -303.572,Z 936.708,A 0.000,B 0.000,C 90.000,E1 127.443} C_DIS
LIN {X -0.066,Y -307.243,Z 936.706,A 0.000,B 0.000,C 90.000,E1 127.076} C_DIS
LIN {X -0.059,Y -310.756,Z 936.703,A 0.000,B 0.000,C 90.000,E1 126.503} C_DIS
LIN {X -0.026,Y -312.166,Z 936.701,A 0.000,B 0.000,C 90.000,E1 126.171} C_DIS
LIN {X 0.075,Y -317.248,Z 936.692,A 0.000,B 0.000,C 90.000,E1 124.532} C_DIS
LIN {X 0.099,Y -328.242,Z 936.674,A 0.000,B 0.000,C 90.000,E1 121.337} C_DIS
LIN {X -0.006,Y -339.522,Z 936.659,A 0.000,B 0.000,C 90.000,E1 118.537} C_DIS
LIN {X 0.009,Y -352.220,Z 936.643,A 0.000,B 0.000,C 90.000,E1 115.771} C_DIS
LIN {X -0.134,Y -364.785,Z 936.630,A 0.000,B 0.000,C 90.000,E1 113.387} C_DIS
LIN {X -0.108,Y -378.646,Z 936.617,A 0.000,B 0.000,C 90.000,E1 111.025} C_DIS
LIN {X -0.140,Y -393.902,Z 936.604,A 0.000,B 0.000,C 90.000,E1 108.725} C_DIS
LIN {X 0.100,Y -410.661,Z 936.591,A 0.000,B 0.000,C 90.000,E1 106.441} C_DIS
LIN {X 0.143,Y -429.045,Z 936.579,A 0.000,B 0.000,C 90.000,E1 104.245} C_DIS
LIN {X -0.077,Y -448.857,Z 936.568,A 0.000,B 0.000,C 90.000,E1 102.175} C_DIS
LIN {X -0.165,Y -466.689,Z 936.558,A 0.000,B 0.000,C 90.000,E1 100.489} C_DIS
LIN {X -0.147,Y -468.884,Z 936.557,A 0.000,B 0.000,C 90.000,E1 100.254} C_DIS
LIN {X 0.162,Y -470.669,Z 936.555,A 0.000,B 0.000,C 90.000,E1 99.962} C_DIS
LIN {X 0.008,Y -472.009,Z 936.554,A 0.000,B 0.000,C 90.000,E1 99.726} C_DIS
LIN {X 0.108,Y -473.689,Z 936.551,A 0.000,B 0.000,C 90.000,E1 99.208} C_DIS
LIN {X -0.249,Y -474.301,Z 936.548,A 0.000,B 0.000,C 90.000,E1 98.746} C_DIS
LIN {X -0.057,Y -473.948,Z 936.546,A 0.000,B 0.000,C 90.000,E1 98.219} C_DIS
LIN {X 0.069,Y -472.581,Z 936.543,A 0.000,B 0.000,C 90.000,E1 97.701} C_DIS
LIN {X -0.073,Y -471.449,Z 936.541,A 0.000,B 0.000,C 90.000,E1 97.466} C_DIS
LIN {X 0.142,Y -464.997,Z 936.536,A 0.000,B 0.000,C 90.000,E1 96.429} C_DIS
LIN {X 0.067,Y -450.506,Z 936.523,A 0.000,B 0.000,C 90.000,E1 94.131} C_DIS
LIN {X 0.140,Y -439.120,Z 936.513,A 0.000,B 0.000,C 90.000,E1 92.293} C_DIS
LIN {X -0.188,Y -424.543,Z 936.500,A 0.000,B 0.000,C 90.000,E1 89.943} C_DIS
LIN {X 0.035,Y -409.018,Z 936.484,A 0.000,B 0.000,C 90.000,E1 87.192} C_DIS
LIN {X 0.092,Y -398.104,Z 936.474,A 0.000,B 0.000,C 90.000,E1 85.241} C_DIS
LIN {X -0.001,Y -387.181,Z 936.463,A 0.000,B 0.000,C 90.000,E1 83.280} C_DIS
LIN {X 0.097,Y -377.643,Z 936.453,A 0.000,B 0.000,C 90.000,E1 81.546} C_DIS
LIN {X 0.078,Y -367.933,Z 936.443,A 0.000,B 0.000,C 90.000,E1 79.803} C_DIS
LIN {X -0.047,Y -358.040,Z 936.434,A 0.000,B 0.000,C 90.000,E1 78.049} C_DIS
LIN {X 0.002,Y -346.236,Z 936.422,A 0.000,B 0.000,C 90.000,E1 75.936} C_DIS
LIN {X 0.007,Y -328.484,Z 936.403,A 0.000,B 0.000,C 90.000,E1 72.543} C_DIS
LIN {X 0.098,Y -317.955,Z 936.391,A 0.000,B 0.000,C 90.000,E1 70.315} C_DIS
LIN {X 0.076,Y -306.077,Z 936.376,A 0.000,B 0.000,C 90.000,E1 67.741} C_DIS
LIN {X -0.151,Y -295.606,Z 936.364,A 0.000,B 0.000,C 90.000,E1 65.485} C_DIS
LIN {X 0.148,Y -283.721,Z 936.349,A 0.000,B 0.000,C 90.000,E1 62.743} C_DIS
LIN {X 0.023,Y -274.720,Z 936.337,A 0.000,B 0.000,C 90.000,E1 60.717} C_DIS
LIN {X -0.012,Y -261.491,Z 936.320,A 0.000,B 0.000,C 90.000,E1 57.582} C_DIS
LIN {X 0.007,Y -249.132,Z 936.302,A 0.000,B 0.000,C 90.000,E1 54.356} C_DIS
LIN {X 0.050,Y -237.959,Z 936.284,A 0.000,B 0.000,C 90.000,E1 51.045} C_DIS
LIN {X 0.032,Y -227.662,Z 936.265,A 0.000,B 0.000,C 90.000,E1 47.676} C_DIS
LIN {X -0.017,Y -219.194,Z 936.248,A 0.000,B 0.000,C 90.000,E1 44.636} C_DIS
LIN {X 0.041,Y -211.403,Z 936.231,A 0.000,B 0.000,C 90.000,E1 41.515} C_DIS
LIN {X -0.049,Y -204.202,Z 936.213,A 0.000,B 0.000,C 90.000,E1 38.382} C_DIS
LIN {X 0.038,Y -197.504,Z 936.195,A 0.000,B 0.000,C 90.000,E1 35.152} C_DIS
LIN {X -0.058,Y -191.323,Z 936.177,A 0.000,B 0.000,C 90.000,E1 31.926} C_DIS
LIN {X -0.014,Y -185.836,Z 936.159,A 0.000,B 0.000,C 90.000,E1 28.615} C_DIS
LIN {X -0.037,Y -180.915,Z 936.140,A 0.000,B 0.000,C 90.000,E1 25.283} C_DIS
LIN {X -0.004,Y -176.750,Z 936.122,A 0.000,B 0.000,C 90.000,E1 21.897} C_DIS
LIN {X -0.018,Y -172.425,Z 936.098,A 0.000,B 0.000,C 90.000,E1 17.638} C_DIS
LIN {X 0.079,Y -169.226,Z 936.074,A 0.000,B 0.000,C 90.000,E1 13.300} C_DIS
LIN {X 0.042,Y -166.799,Z 936.045,A 0.000,B 0.000,C 90.000,E1 8.106} C_DIS
LIN {X -0.030,Y -167.147,Z 935.973,A 0.000,B 0.000,C 90.000,E1 355.179} C_DIS
LIN {X -0.085,Y -169.873,Z 935.944,A 0.000,B 0.000,C 90.000,E1 349.982} C_DIS
LIN {X -0.027,Y -173.311,Z 935.920,A 0.000,B 0.000,C 90.000,E1 345.644} C_DIS
LIN {X 0.080,Y -176.829,Z 935.901,A 0.000,B 0.000,C 90.000,E1 342.181} C_DIS
LIN {X 0.108,Y -181.001,Z 935.882,A 0.000,B 0.000,C 90.000,E1 338.773} C_DIS
LIN {X 0.026,Y -185.852,Z 935.864,A 0.000,B 0.000,C 90.000,E1 335.433} C_DIS
LIN {X 0.031,Y -191.466,Z 935.845,A 0.000,B 0.000,C 90.000,E1 332.103} C_DIS
LIN {X 0.020,Y -197.808,Z 935.827,A 0.000,B 0.000,C 90.000,E1 328.820} C_DIS
LIN {X -0.030,Y -204.697,Z 935.809,A 0.000,B 0.000,C 90.000,E1 325.595} C_DIS
LIN {X -0.002,Y -212.168,Z 935.791,A 0.000,B 0.000,C 90.000,E1 322.396} C_DIS
LIN {X 0.074,Y -221.165,Z 935.771,A 0.000,B 0.000,C 90.000,E1 318.852} C_DIS
LIN {X -0.046,Y -230.093,Z 935.754,A 0.000,B 0.000,C 90.000,E1 315.810} C_DIS
LIN {X 0.059,Y -240.080,Z 935.738,A 0.000,B 0.000,C 90.000,E1 312.771} C_DIS
LIN {X -0.073,Y -251.197,Z 935.721,A 0.000,B 0.000,C 90.000,E1 309.850} C_DIS
LIN {X -0.010,Y -263.895,Z 935.705,A 0.000,B 0.000,C 90.000,E1 306.950} C_DIS
LIN {X -0.012,Y -276.384,Z 935.692,A 0.000,B 0.000,C 90.000,E1 304.485} C_DIS
LIN {X 0.073,Y -294.008,Z 935.674,A 0.000,B 0.000,C 90.000,E1 301.386} C_DIS
LIN {X 0.045,Y -313.181,Z 935.658,A 0.000,B 0.000,C 90.000,E1 298.409} C_DIS
LIN {X -0.011,Y -327.366,Z 935.647,A 0.000,B 0.000,C 90.000,E1 296.488} C_DIS
LIN {X 0.089,Y -350.562,Z 935.632,A 0.000,B 0.000,C 90.000,E1 293.695} C_DIS
LIN {X -0.176,Y -369.259,Z 935.620,A 0.000,B 0.000,C 90.000,E1 291.716} C_DIS
LIN {X -0.021,Y -385.078,Z 935.611,A 0.000,B 0.000,C 90.000,E1 290.066} C_DIS
LIN {X 0.013,Y -398.128,Z 935.604,A 0.000,B 0.000,C 90.000,E1 288.725} C_DIS
LIN {X -0.118,Y -410.977,Z 935.597,A 0.000,B 0.000,C 90.000,E1 287.402} C_DIS
LIN {X -0.076,Y -421.027,Z 935.591,A 0.000,B 0.000,C 90.000,E1 286.315} C_DIS
LIN {X -0.190,Y -430.638,Z 935.585,A 0.000,B 0.000,C 90.000,E1 285.245} C_DIS
LIN {X 0.224,Y -439.610,Z 935.579,A 0.000,B 0.000,C 90.000,E1 284.120} C_DIS
LIN {X 0.022,Y -450.422,Z 935.571,A 0.000,B 0.000,C 90.000,E1 282.827} C_DIS
LIN {X 0.147,Y -458.575,Z 935.565,A 0.000,B 0.000,C 90.000,E1 281.771} C_DIS
LIN {X -0.175,Y -466.241,Z 935.560,A 0.000,B 0.000,C 90.000,E1 280.782} C_DIS
LIN {X 0.133,Y -473.320,Z 935.554,A 0.000,B 0.000,C 90.000,E1 279.726} C_DIS
LIN {X 0.101,Y -478.107,Z 935.550,A 0.000,B 0.000,C 90.000,E1 278.973} C_DIS
LIN {X 0.117,Y -482.128,Z 935.546,A 0.000,B 0.000,C 90.000,E1 278.219} C_DIS
LIN {X 0.100,Y -485.463,Z 935.542,A 0.000,B 0.000,C 90.000,E1 277.473} C_DIS
LIN {X -0.132,Y -487.300,Z 935.539,A 0.000,B 0.000,C 90.000,E1 277.004} C_DIS
LIN {X 0.063,Y -488.839,Z 935.536,A 0.000,B 0.000,C 90.000,E1 276.486} C_DIS
LIN {X -0.218,Y -490.069,Z 935.533,A 0.000,B 0.000,C 90.000,E1 276.024} C_DIS
LIN {X -0.051,Y -490.938,Z 935.531,A 0.000,B 0.000,C 90.000,E1 275.511} C_DIS
LIN {X 0.173,Y -491.423,Z 935.528,A 0.000,B 0.000,C 90.000,E1 274.992} C_DIS
LIN {X -0.089,Y -491.544,Z 935.525,A 0.000,B 0.000,C 90.000,E1 274.531} C_DIS
LIN {X 0.139,Y -491.182,Z 935.522,A 0.000,B 0.000,C 90.000,E1 274.012} C_DIS
LIN {X -0.156,Y -490.328,Z 935.520,A 0.000,B 0.000,C 90.000,E1 273.555} C_DIS
LIN {X 0.066,Y -488.945,Z 935.517,A 0.000,B 0.000,C 90.000,E1 273.037} C_DIS
LIN {X -0.229,Y -486.900,Z 935.514,A 0.000,B 0.000,C 90.000,E1 272.579} C_DIS
LIN {X -0.043,Y -484.172,Z 935.511,A 0.000,B 0.000,C 90.000,E1 272.064} C_DIS
LIN {X -0.185,Y -482.558,Z 935.510,A 0.000,B 0.000,C 90.000,E1 271.833} C_DIS
LIN {X -0.028,Y -478.580,Z 935.507,A 0.000,B 0.000,C 90.000,E1 271.318} C_DIS
LIN {X 0.108,Y -473.631,Z 935.505,A 0.000,B 0.000,C 90.000,E1 270.802} C_DIS
LIN {X -0.041,Y -467.894,Z 935.502,A 0.000,B 0.000,C 90.000,E1 270.344} C_DIS
LIN {X 0.210,Y -461.801,Z 935.500,A 0.000,B 0.000,C 90.000,E1 269.885} C_DIS
LIN {X -0.022,Y -455.382,Z 935.497,A 0.000,B 0.000,C 90.000,E1 269.542} C_DIS
LIN {X 0.156,Y -448.759,Z 935.496,A 0.000,B 0.000,C 90.000,E1 269.198} C_DIS
LIN {X 0.204,Y -441.830,Z 935.494,A 0.000,B 0.000,C 90.000,E1 268.912} C_DIS
LIN {X 0.120,Y -434.684,Z 935.493,A 0.000,B 0.000,C 90.000,E1 268.682} C_DIS
LIN {X -0.066,Y -427.239,Z 935.492,A 0.000,B 0.000,C 90.000,E1 268.511} C_DIS
LIN {X 0.073,Y -419.453,Z 935.491,A 0.000,B 0.000,C 90.000,E1 268.339} C_DIS
LIN {X 0.083,Y -410.247,Z 935.490,A 0.000,B 0.000,C 90.000,E1 268.224} C_DIS
LIN {X -0.125,Y -404.712,Z 935.490,A 0.000,B 0.000,C 90.000,E1 268.224} C_DIS
LIN {X -0.075,Y -181.158,Z 935.490,A 0.000,B 0.000,C 90.000,E1 268.224} C_DIS
LIN {X -0.093,Y -180.905,Z 935.474,A 0.000,B 0.000,C 90.000,E1 265.355} C_DIS
LIN {X -0.018,Y -180.667,Z 935.469,A 0.000,B 0.000,C 90.000,E1 264.489} C_DIS
LIN {X 0.056,Y -178.747,Z 935.441,A 0.000,B 0.000,C 90.000,E1 259.398} C_DIS
LIN {X -0.047,Y -175.795,Z 935.413,A 0.000,B 0.000,C 90.000,E1 254.338} C_DIS
LIN {X -0.052,Y -171.980,Z 935.384,A 0.000,B 0.000,C 90.000,E1 249.209} C_DIS
LIN {X -0.014,Y -171.385,Z 935.380,A 0.000,B 0.000,C 90.000,E1 248.337} C_DIS
LIN {X -0.028,Y -167.629,Z 935.356,A 0.000,B 0.000,C 90.000,E1 244.024} C_DIS
LIN {X -0.013,Y -166.284,Z 935.346,A 0.000,B 0.000,C 90.000,E1 242.281} C_DIS
LIN {X -0.019,Y -163.032,Z 935.327,A 0.000,B 0.000,C 90.000,E1 238.791} C_DIS
LIN {X 0.033,Y -160.961,Z 935.312,A 0.000,B 0.000,C 90.000,E1 236.135} C_DIS
LIN {X -0.079,Y -157.715,Z 935.292,A 0.000,B 0.000,C 90.000,E1 232.637} C_DIS
LIN {X 0.080,Y -155.755,Z 935.277,A 0.000,B 0.000,C 90.000,E1 229.908} C_DIS
LIN {X -0.083,Y -152.011,Z 935.253,A 0.000,B 0.000,C 90.000,E1 225.486} C_DIS
LIN {X -0.064,Y -150.258,Z 935.237,A 0.000,B 0.000,C 90.000,E1 222.771} C_DIS
LIN {X 0.069,Y -147.012,Z 935.212,A 0.000,B 0.000,C 90.000,E1 218.177} C_DIS
LIN {X 0.059,Y -145.595,Z 935.197,A 0.000,B 0.000,C 90.000,E1 215.438} C_DIS
LIN {X -0.021,Y -142.983,Z 935.172,A 0.000,B 0.000,C 90.000,E1 210.875} C_DIS
LIN {X -0.020,Y -141.610,Z 935.151,A 0.000,B 0.000,C 90.000,E1 207.180} C_DIS
LIN {X 0.021,Y -139.427,Z 935.115,A 0.000,B 0.000,C 90.000,E1 200.663} C_DIS
LIN {X 0.072,Y -139.156,Z 935.104,A 0.000,B 0.000,C 90.000,E1 198.779} C_DIS
LIN {X -0.042,Y -138.343,Z 935.058,A 0.000,B 0.000,C 90.000,E1 190.423} C_DIS
LIN {X -0.061,Y -139.482,Z 935.006,A 0.000,B 0.000,C 90.000,E1 181.088} C_DIS
LIN {X 0.021,Y -141.075,Z 934.975,A 0.000,B 0.000,C 90.000,E1 175.469} C_DIS
LIN {X -0.026,Y -142.451,Z 934.959,A 0.000,B 0.000,C 90.000,E1 172.704} C_DIS
LIN {X 0.064,Y -144.693,Z 934.934,A 0.000,B 0.000,C 90.000,E1 168.049} C_DIS
LIN {X 0.016,Y -147.286,Z 934.913,A 0.000,B 0.000,C 90.000,E1 164.393} C_DIS
LIN {X 0.033,Y -150.605,Z 934.888,A 0.000,B 0.000,C 90.000,E1 159.826} C_DIS
LIN {X -0.031,Y -154.080,Z 934.868,A 0.000,B 0.000,C 90.000,E1 156.230} C_DIS
LIN {X 0.034,Y -157.499,Z 934.848,A 0.000,B 0.000,C 90.000,E1 152.615} C_DIS
LIN {X -0.020,Y -161.729,Z 934.828,A 0.000,B 0.000,C 90.000,E1 149.076} C_DIS
LIN {X -0.007,Y -165.923,Z 934.809,A 0.000,B 0.000,C 90.000,E1 145.548} C_DIS
LIN {X -0.020,Y -170.910,Z 934.789,A 0.000,B 0.000,C 90.000,E1 142.065} C_DIS
LIN {X 0.006,Y -175.777,Z 934.770,A 0.000,B 0.000,C 90.000,E1 138.609} C_DIS
LIN {X 0.007,Y -181.387,Z 934.751,A 0.000,B 0.000,C 90.000,E1 135.202} C_DIS
LIN {X 0.010,Y -186.883,Z 934.732,A 0.000,B 0.000,C 90.000,E1 131.838} C_DIS
LIN {X -0.037,Y -191.466,Z 934.719,A 0.000,B 0.000,C 90.000,E1 129.358} C_DIS
LIN {X 0.106,Y -194.166,Z 934.710,A 0.000,B 0.000,C 90.000,E1 127.729} C_DIS
LIN {X 0.127,Y -296.773,Z 934.710,A 0.000,B 0.000,C 90.000,E1 127.729} C_DIS
LIN {X -0.163,Y -299.273,Z 934.709,A 0.000,B 0.000,C 90.000,E1 127.729} C_DIS
LIN {X 0.018,Y -302.634,Z 934.708,A 0.000,B 0.000,C 90.000,E1 127.523} C_DIS
LIN {X -0.139,Y -306.155,Z 934.707,A 0.000,B 0.000,C 90.000,E1 127.237} C_DIS
LIN {X -0.091,Y -309.762,Z 934.704,A 0.000,B 0.000,C 90.000,E1 126.710} C_DIS
LIN {X -0.063,Y -311.365,Z 934.702,A 0.000,B 0.000,C 90.000,E1 126.377} C_DIS
LIN {X 0.151,Y -312.625,Z 934.700,A 0.000,B 0.000,C 90.000,E1 126.011} C_DIS
LIN {X 0.017,Y -324.067,Z 934.681,A 0.000,B 0.000,C 90.000,E1 122.498} C_DIS
LIN {X -0.035,Y -334.810,Z 934.665,A 0.000,B 0.000,C 90.000,E1 119.667} C_DIS
LIN {X 0.014,Y -346.924,Z 934.649,A 0.000,B 0.000,C 90.000,E1 116.873} C_DIS
LIN {X 0.093,Y -360.523,Z 934.634,A 0.000,B 0.000,C 90.000,E1 114.131} C_DIS
LIN {X 0.018,Y -373.951,Z 934.621,A 0.000,B 0.000,C 90.000,E1 111.770} C_DIS
LIN {X 0.005,Y -388.739,Z 934.608,A 0.000,B 0.000,C 90.000,E1 109.450} C_DIS
LIN {X 0.119,Y -404.994,Z 934.595,A 0.000,B 0.000,C 90.000,E1 107.166} C_DIS
LIN {X 0.137,Y -422.834,Z 934.583,A 0.000,B 0.000,C 90.000,E1 104.954} C_DIS
LIN {X 0.026,Y -442.292,Z 934.571,A 0.000,B 0.000,C 90.000,E1 102.827} C_DIS
LIN {X 0.067,Y -462.540,Z 934.560,A 0.000,B 0.000,C 90.000,E1 100.838} C_DIS
LIN {X 0.081,Y -467.614,Z 934.558,A 0.000,B 0.000,C 90.000,E1 100.366} C_DIS
LIN {X -0.018,Y -469.604,Z 934.556,A 0.000,B 0.000,C 90.000,E1 100.141} C_DIS
LIN {X -0.035,Y -471.116,Z 934.555,A 0.000,B 0.000,C 90.000,E1 99.905} C_DIS
LIN {X -0.182,Y -472.337,Z 934.554,A 0.000,B 0.000,C 90.000,E1 99.670} C_DIS
LIN {X 0.137,Y -473.231,Z 934.552,A 0.000,B 0.000,C 90.000,E1 99.378} C_DIS
LIN {X -0.220,Y -474.191,Z 934.549,A 0.000,B 0.000,C 90.000,E1 98.916} C_DIS
LIN {X -0.101,Y -474.171,Z 934.547,A 0.000,B 0.000,C 90.000,E1 98.398} C_DIS
LIN {X 0.091,Y -473.172,Z 934.544,A 0.000,B 0.000,C 90.000,E1 97.871} C_DIS
LIN {X 0.214,Y -471.024,Z 934.541,A 0.000,B 0.000,C 90.000,E1 97.352} C_DIS
LIN {X 0.102,Y -458.029,Z 934.530,A 0.000,B 0.000,C 90.000,E1 95.334} C_DIS
LIN {X 0.121,Y -448.460,Z 934.521,A 0.000,B 0.000,C 90.000,E1 93.784} C_DIS
LIN {X -0.126,Y -435.461,Z 934.509,A 0.000,B 0.000,C 90.000,E1 91.718} C_DIS
LIN {X -0.013,Y -419.394,Z 934.495,A 0.000,B 0.000,C 90.000,E1 89.026} C_DIS
LIN {X -0.163,Y -408.592,Z 934.484,A 0.000,B 0.000,C 90.000,E1 87.135} C_DIS
LIN {X -0.072,Y -397.674,Z 934.473,A 0.000,B 0.000,C 90.000,E1 85.179} C_DIS
LIN {X 0.176,Y -386.719,Z 934.462,A 0.000,B 0.000,C 90.000,E1 83.166} C_DIS
LIN {X -0.114,Y -377.189,Z 934.453,A 0.000,B 0.000,C 90.000,E1 81.489} C_DIS
LIN {X -0.131,Y -369.093,Z 934.445,A 0.000,B 0.000,C 90.000,E1 80.038} C_DIS
LIN {X 0.120,Y -359.226,Z 934.435,A 0.000,B 0.000,C 90.000,E1 78.229} C_DIS
LIN {X -0.153,Y -347.451,Z 934.423,A 0.000,B 0.000,C 90.000,E1 76.172} C_DIS
LIN {X -0.098,Y -329.603,Z 934.404,A 0.000,B 0.000,C 90.000,E1 72.779} C_DIS
LIN {X -0.032,Y -317.528,Z 934.390,A 0.000,B 0.000,C 90.000,E1 70.242} C_DIS
LIN {X -0.050,Y -305.668,Z 934.376,A 0.000,B 0.000,C 90.000,E1 67.667} C_DIS
LIN {X -0.011,Y -295.196,Z 934.363,A 0.000,B 0.000,C 90.000,E1 65.357} C_DIS
LIN {X 0.050,Y -284.789,Z 934.350,A 0.000,B 0.000,C 90.000,E1 62.999} C_DIS
LIN {X -0.052,Y -275.802,Z 934.339,A 0.000,B 0.000,C 90.000,E1 60.973} C_DIS
LIN {X -0.050,Y -262.492,Z 934.321,A 0.000,B 0.000,C 90.000,E1 57.837} C_DIS
LIN {X 0.006,Y -250.036,Z 934.303,A 0.000,B 0.000,C 90.000,E1 54.609} C_DIS
LIN {X -0.064,Y -238.801,Z 934.285,A 0.000,B 0.000,C 90.000,E1 51.331} C_DIS
LIN {X -0.036,Y -228.469,Z 934.266,A 0.000,B 0.000,C 90.000,E1 47.957} C_DIS
LIN {X -0.070,Y -219.981,Z 934.249,A 0.000,B 0.000,C 90.000,E1 44.919} C_DIS
LIN {X -0.139,Y -212.164,Z 934.232,A 0.000,B 0.000,C 90.000,E1 41.838} C_DIS
LIN {X -0.072,Y -204.959,Z 934.215,A 0.000,B 0.000,C 90.000,E1 38.669} C_DIS
LIN {X 0.033,Y -198.224,Z 934.197,A 0.000,B 0.000,C 90.000,E1 35.438} C_DIS
LIN {X -0.043,Y -192.023,Z 934.179,A 0.000,B 0.000,C 90.000,E1 32.212} C_DIS
LIN {X 0.024,Y -186.472,Z 934.161,A 0.000,B 0.000,C 90.000,E1 28.899} C_DIS
LIN {X -0.061,Y -181.516,Z 934.142,A 0.000,B 0.000,C 90.000,E1 25.591} C_DIS
LIN {X -0.015,Y -177.281,Z 934.123,A 0.000,B 0.000,C 90.000,E1 22.206} C_DIS
LIN {X -0.012,Y -172.899,Z 934.100,A 0.000,B 0.000,C 90.000,E1 17.946} C_DIS
LIN {X -0.020,Y -169.630,Z 934.076,A 0.000,B 0.000,C 90.000,E1 13.647} C_DIS
LIN {X -0.043,Y -167.113,Z 934.047,A 0.000,B 0.000,C 90.000,E1 8.454} C_DIS
LIN {X -0.023,Y -167.383,Z 933.973,A 0.000,B 0.000,C 90.000,E1 355.179} C_DIS
LIN {X -0.069,Y -170.134,Z 933.944,A 0.000,B 0.000,C 90.000,E1 349.982} C_DIS
LIN {X -0.002,Y -173.557,Z 933.920,A 0.000,B 0.000,C 90.000,E1 345.644} C_DIS
LIN {X -0.058,Y -177.072,Z 933.901,A 0.000,B 0.000,C 90.000,E1 342.236} C_DIS
LIN {X -0.023,Y -181.244,Z 933.882,A 0.000,B 0.000,C 90.000,E1 338.827} C_DIS
LIN {X -0.098,Y -186.101,Z 933.864,A 0.000,B 0.000,C 90.000,E1 335.485} C_DIS
LIN {X -0.085,Y -191.735,Z 933.845,A 0.000,B 0.000,C 90.000,E1 332.153} C_DIS
LIN {X -0.088,Y -198.080,Z 933.827,A 0.000,B 0.000,C 90.000,E1 328.869} C_DIS
LIN {X 0.040,Y -204.963,Z 933.809,A 0.000,B 0.000,C 90.000,E1 325.595} C_DIS
LIN {X 0.077,Y -212.423,Z 933.791,A 0.000,B 0.000,C 90.000,E1 322.396} C_DIS
LIN {X -0.068,Y -220.383,Z 933.774,A 0.000,B 0.000,C 90.000,E1 319.299} C_DIS
LIN {X -0.044,Y -229.191,Z 933.757,A 0.000,B 0.000,C 90.000,E1 316.215} C_DIS
LIN {X 0.036,Y -239.012,Z 933.740,A 0.000,B 0.000,C 90.000,E1 313.176} C_DIS
LIN {X 0.043,Y -249.947,Z 933.723,A 0.000,B 0.000,C 90.000,E1 310.216} C_DIS
LIN {X 0.077,Y -262.398,Z 933.707,A 0.000,B 0.000,C 90.000,E1 307.317} C_DIS
LIN {X -0.098,Y -272.795,Z 933.696,A 0.000,B 0.000,C 90.000,E1 305.231} C_DIS
LIN {X -0.130,Y -289.976,Z 933.678,A 0.000,B 0.000,C 90.000,E1 302.133} C_DIS
LIN {X 0.136,Y -308.697,Z 933.662,A 0.000,B 0.000,C 90.000,E1 299.077} C_DIS
LIN {X 0.082,Y -319.971,Z 933.653,A 0.000,B 0.000,C 90.000,E1 297.462} C_DIS
LIN {X -0.131,Y -334.713,Z 933.642,A 0.000,B 0.000,C 90.000,E1 295.591} C_DIS
LIN {X -0.142,Y -358.057,Z 933.627,A 0.000,B 0.000,C 90.000,E1 292.898} C_DIS
LIN {X -0.144,Y -376.767,Z 933.616,A 0.000,B 0.000,C 90.000,E1 290.918} C_DIS
LIN {X 0.114,Y -390.022,Z 933.609,A 0.000,B 0.000,C 90.000,E1 289.523} C_DIS
LIN {X 0.129,Y -402.994,Z 933.601,A 0.000,B 0.000,C 90.000,E1 288.181} C_DIS
LIN {X -0.032,Y -415.740,Z 933.594,A 0.000,B 0.000,C 90.000,E1 286.858} C_DIS
LIN {X -0.041,Y -425.528,Z 933.588,A 0.000,B 0.000,C 90.000,E1 285.788} C_DIS
LIN {X -0.105,Y -434.831,Z 933.582,A 0.000,B 0.000,C 90.000,E1 284.717} C_DIS
LIN {X 0.156,Y -445.865,Z 933.574,A 0.000,B 0.000,C 90.000,E1 283.355} C_DIS
LIN {X -0.214,Y -454.257,Z 933.568,A 0.000,B 0.000,C 90.000,E1 282.355} C_DIS
LIN {X -0.050,Y -462.219,Z 933.563,A 0.000,B 0.000,C 90.000,E1 281.299} C_DIS
LIN {X 0.124,Y -469.580,Z 933.557,A 0.000,B 0.000,C 90.000,E1 280.254} C_DIS
LIN {X 0.062,Y -474.775,Z 933.553,A 0.000,B 0.000,C 90.000,E1 279.500} C_DIS
LIN {X 0.051,Y -479.334,Z 933.549,A 0.000,B 0.000,C 90.000,E1 278.746} C_DIS
LIN {X 0.077,Y -483.200,Z 933.544,A 0.000,B 0.000,C 90.000,E1 277.992} C_DIS
LIN {X -0.228,Y -485.358,Z 933.542,A 0.000,B 0.000,C 90.000,E1 277.530} C_DIS
LIN {X 0.022,Y -487.237,Z 933.539,A 0.000,B 0.000,C 90.000,E1 277.004} C_DIS
LIN {X 0.217,Y -488.804,Z 933.536,A 0.000,B 0.000,C 90.000,E1 276.486} C_DIS
LIN {X -0.116,Y -490.020,Z 933.533,A 0.000,B 0.000,C 90.000,E1 276.030} C_DIS
LIN {X 0.102,Y -490.921,Z 933.531,A 0.000,B 0.000,C 90.000,E1 275.511} C_DIS
LIN {X -0.162,Y -491.427,Z 933.528,A 0.000,B 0.000,C 90.000,E1 275.049} C_DIS
LIN {X 0.065,Y -491.581,Z 933.525,A 0.000,B 0.000,C 90.000,E1 274.531} C_DIS
LIN {X -0.198,Y -491.259,Z 933.522,A 0.000,B 0.000,C 90.000,E1 274.069} C_DIS
LIN {X -0.003,Y -490.456,Z 933.520,A 0.000,B 0.000,C 90.000,E1 273.555} C_DIS
LIN {X 0.220,Y -489.087,Z 933.517,A 0.000,B 0.000,C 90.000,E1 273.037} C_DIS
LIN {X -0.075,Y -487.122,Z 933.514,A 0.000,B 0.000,C 90.000,E1 272.579} C_DIS
LIN {X 0.111,Y -484.441,Z 933.512,A 0.000,B 0.000,C 90.000,E1 272.064} C_DIS
LIN {X -0.189,Y -480.965,Z 933.509,A 0.000,B 0.000,C 90.000,E1 271.604} C_DIS
LIN {X -0.038,Y -476.629,Z 933.506,A 0.000,B 0.000,C 90.000,E1 271.088} C_DIS
LIN {X 0.089,Y -471.247,Z 933.503,A 0.000,B 0.000,C 90.000,E1 270.573} C_DIS
LIN {X 0.094,Y -465.294,Z 933.501,A 0.000,B 0.000,C 90.000,E1 270.115} C_DIS
LIN {X 0.073,Y -459.044,Z 933.498,A 0.000,B 0.000,C 90.000,E1 269.714} C_DIS
LIN {X -0.005,Y -452.402,Z 933.497,A 0.000,B 0.000,C 90.000,E1 269.370} C_DIS
LIN {X -0.108,Y -445.775,Z 933.495,A 0.000,B 0.000,C 90.000,E1 269.083} C_DIS
LIN {X 0.079,Y -438.752,Z 933.493,A 0.000,B 0.000,C 90.000,E1 268.797} C_DIS
LIN {X 0.165,Y -431.678,Z 933.492,A 0.000,B 0.000,C 90.000,E1 268.568} C_DIS
LIN {X 0.047,Y -423.786,Z 933.491,A 0.000,B 0.000,C 90.000,E1 268.396} C_DIS
LIN {X -0.140,Y -414.690,Z 933.490,A 0.000,B 0.000,C 90.000,E1 268.282} C_DIS
LIN {X 0.171,Y -406.125,Z 933.490,A 0.000,B 0.000,C 90.000,E1 268.167} C_DIS
LIN {X 0.141,Y -402.985,Z 933.490,A 0.000,B 0.000,C 90.000,E1 268.165} C_DIS
LIN {X 0.045,Y -181.154,Z 933.490,A 0.000,B 0.000,C 90.000,E1 268.165} C_DIS
LIN {X 0.020,Y -180.904,Z 933.474,A 0.000,B 0.000,C 90.000,E1 265.298} C_DIS
LIN {X -0.030,Y -180.247,Z 933.465,A 0.000,B 0.000,C 90.000,E1 263.628} C_DIS
LIN {X -0.011,Y -178.734,Z 933.441,A 0.000,B 0.000,C 90.000,E1 259.398} C_DIS
LIN {X 0.056,Y -175.782,Z 933.413,A 0.000,B 0.000,C 90.000,E1 254.283} C_DIS
LIN {X 0.043,Y -171.967,Z 933.384,A 0.000,B 0.000,C 90.000,E1 249.156} C_DIS
LIN {X 0.080,Y -171.364,Z 933.380,A 0.000,B 0.000,C 90.000,E1 248.284} C_DIS
LIN {X -0.093,Y -167.612,Z 933.356,A 0.000,B 0.000,C 90.000,E1 244.024} C_DIS
LIN {X 0.070,Y -166.261,Z 933.346,A 0.000,B 0.000,C 90.000,E1 242.231} C_DIS
LIN {X 0.057,Y -163.014,Z 933.326,A 0.000,B 0.000,C 90.000,E1 238.742} C_DIS
LIN {X -0.030,Y -160.939,Z 933.312,A 0.000,B 0.000,C 90.000,E1 236.135} C_DIS
LIN {X 0.080,Y -157.697,Z 933.292,A 0.000,B 0.000,C 90.000,E1 232.557} C_DIS
LIN {X 0.018,Y -155.736,Z 933.277,A 0.000,B 0.000,C 90.000,E1 229.908} C_DIS
LIN {X 0.071,Y -151.994,Z 933.252,A 0.000,B 0.000,C 90.000,E1 225.405} C_DIS
LIN {X 0.087,Y -150.239,Z 933.237,A 0.000,B 0.000,C 90.000,E1 222.690} C_DIS
LIN {X 0.009,Y -146.998,Z 933.212,A 0.000,B 0.000,C 90.000,E1 218.177} C_DIS
LIN {X 0.000,Y -145.584,Z 933.197,A 0.000,B 0.000,C 90.000,E1 215.438} C_DIS
LIN {X -0.006,Y -142.972,Z 933.171,A 0.000,B 0.000,C 90.000,E1 210.846} C_DIS
LIN {X 0.046,Y -141.598,Z 933.151,A 0.000,B 0.000,C 90.000,E1 207.129} C_DIS
LIN {X -0.037,Y -139.423,Z 933.115,A 0.000,B 0.000,C 90.000,E1 200.663} C_DIS
LIN {X 0.014,Y -139.150,Z 933.104,A 0.000,B 0.000,C 90.000,E1 198.779} C_DIS
LIN {X 0.036,Y -138.346,Z 933.058,A 0.000,B 0.000,C 90.000,E1 190.366} C_DIS
LIN {X 0.021,Y -139.486,Z 933.006,A 0.000,B 0.000,C 90.000,E1 181.031} C_DIS
LIN {X -0.039,Y -141.086,Z 932.975,A 0.000,B 0.000,C 90.000,E1 175.469} C_DIS
LIN {X 0.057,Y -142.463,Z 932.959,A 0.000,B 0.000,C 90.000,E1 172.648} C_DIS
LIN {X 0.005,Y -144.707,Z 932.934,A 0.000,B 0.000,C 90.000,E1 168.049} C_DIS
LIN {X -0.044,Y -147.305,Z 932.913,A 0.000,B 0.000,C 90.000,E1 164.393} C_DIS
LIN {X -0.030,Y -150.625,Z 932.888,A 0.000,B 0.000,C 90.000,E1 159.826} C_DIS
LIN {X 0.047,Y -154.101,Z 932.868,A 0.000,B 0.000,C 90.000,E1 156.177} C_DIS
LIN {X -0.028,Y -157.524,Z 932.848,A 0.000,B 0.000,C 90.000,E1 152.615} C_DIS
LIN {X -0.084,Y -161.758,Z 932.828,A 0.000,B 0.000,C 90.000,E1 149.076} C_DIS
LIN {X 0.022,Y -165.951,Z 932.808,A 0.000,B 0.000,C 90.000,E1 145.515} C_DIS
LIN {X 0.018,Y -170.943,Z 932.789,A 0.000,B 0.000,C 90.000,E1 142.029} C_DIS
LIN {X -0.061,Y -175.811,Z 932.770,A 0.000,B 0.000,C 90.000,E1 138.609} C_DIS
LIN {X 0.066,Y -181.418,Z 932.751,A 0.000,B 0.000,C 90.000,E1 135.162} C_DIS
LIN {X -0.059,Y -186.922,Z 932.732,A 0.000,B 0.000,C 90.000,E1 131.838} C_DIS
LIN {X 0.013,Y -191.501,Z 932.719,A 0.000,B 0.000,C 90.000,E1 129.322} C_DIS
LIN {X -0.063,Y -194.111,Z 932.710,A 0.000,B 0.000,C 90.000,E1 127.810} C_DIS
LIN {X -0.132,Y -296.255,Z 932.710,A 0.000,B 0.000,C 90.000,E1 127.810} C_DIS
LIN {X -0.036,Y -300.379,Z 932.709,A 0.000,B 0.000,C 90.000,E1 127.684} C_DIS
LIN {X -0.174,Y -303.401,Z 932.708,A 0.000,B 0.000,C 90.000,E1 127.523} C_DIS
LIN {X 0.019,Y -307.087,Z 932.706,A 0.000,B 0.000,C 90.000,E1 127.111} C_DIS
LIN {X 0.016,Y -310.592,Z 932.703,A 0.000,B 0.000,C 90.000,E1 126.537} C_DIS
LIN {X -0.018,Y -311.992,Z 932.701,A 0.000,B 0.000,C 90.000,E1 126.217} C_DIS
LIN {X 0.207,Y -319.126,Z 932.689,A 0.000,B 0.000,C 90.000,E1 123.913} C_DIS
LIN {X 0.020,Y -329.211,Z 932.673,A 0.000,B 0.000,C 90.000,E1 121.082} C_DIS
LIN {X -0.060,Y -340.622,Z 932.657,A 0.000,B 0.000,C 90.000,E1 118.281} C_DIS
LIN {X -0.163,Y -353.456,Z 932.642,A 0.000,B 0.000,C 90.000,E1 115.540} C_DIS
LIN {X -0.124,Y -366.155,Z 932.628,A 0.000,B 0.000,C 90.000,E1 113.131} C_DIS
LIN {X 0.151,Y -380.159,Z 932.615,A 0.000,B 0.000,C 90.000,E1 110.737} C_DIS
LIN {X -0.069,Y -395.569,Z 932.603,A 0.000,B 0.000,C 90.000,E1 108.471} C_DIS
LIN {X 0.092,Y -412.495,Z 932.590,A 0.000,B 0.000,C 90.000,E1 106.205} C_DIS
LIN {X 0.182,Y -431.059,Z 932.578,A 0.000,B 0.000,C 90.000,E1 104.008} C_DIS
LIN {X 0.002,Y -450.954,Z 932.566,A 0.000,B 0.000,C 90.000,E1 101.951} C_DIS
LIN {X 0.101,Y -466.269,Z 932.558,A 0.000,B 0.000,C 90.000,E1 100.489} C_DIS
LIN {X 0.116,Y -468.567,Z 932.557,A 0.000,B 0.000,C 90.000,E1 100.254} C_DIS
LIN {X -0.005,Y -470.402,Z 932.556,A 0.000,B 0.000,C 90.000,E1 100.018} C_DIS
LIN {X -0.129,Y -471.787,Z 932.554,A 0.000,B 0.000,C 90.000,E1 99.782} C_DIS
LIN {X -0.031,Y -473.569,Z 932.551,A 0.000,B 0.000,C 90.000,E1 99.265} C_DIS
LIN {X 0.078,Y -474.266,Z 932.549,A 0.000,B 0.000,C 90.000,E1 98.746} C_DIS
LIN {X -0.199,Y -473.995,Z 932.546,A 0.000,B 0.000,C 90.000,E1 98.276} C_DIS
LIN {X -0.074,Y -472.721,Z 932.543,A 0.000,B 0.000,C 90.000,E1 97.757} C_DIS
LIN {X 0.191,Y -471.646,Z 932.542,A 0.000,B 0.000,C 90.000,E1 97.473} C_DIS
LIN {X -0.098,Y -468.540,Z 932.539,A 0.000,B 0.000,C 90.000,E1 97.004} C_DIS
LIN {X 0.172,Y -452.452,Z 932.525,A 0.000,B 0.000,C 90.000,E1 94.416} C_DIS
LIN {X 0.096,Y -442.791,Z 932.516,A 0.000,B 0.000,C 90.000,E1 92.865} C_DIS
LIN {X -0.008,Y -431.428,Z 932.506,A 0.000,B 0.000,C 90.000,E1 91.031} C_DIS
LIN {X -0.014,Y -415.538,Z 932.491,A 0.000,B 0.000,C 90.000,E1 88.339} C_DIS
LIN {X 0.117,Y -406.251,Z 932.482,A 0.000,B 0.000,C 90.000,E1 86.674} C_DIS
LIN {X 0.119,Y -395.332,Z 932.471,A 0.000,B 0.000,C 90.000,E1 84.723} C_DIS
LIN {X -0.029,Y -384.348,Z 932.460,A 0.000,B 0.000,C 90.000,E1 82.761} C_DIS
LIN {X 0.023,Y -373.191,Z 932.449,A 0.000,B 0.000,C 90.000,E1 80.735} C_DIS
LIN {X -0.100,Y -361.696,Z 932.437,A 0.000,B 0.000,C 90.000,E1 78.701} C_DIS
LIN {X 0.083,Y -351.638,Z 932.427,A 0.000,B 0.000,C 90.000,E1 76.881} C_DIS
LIN {X 0.067,Y -338.312,Z 932.414,A 0.000,B 0.000,C 90.000,E1 74.448} C_DIS
LIN {X 0.059,Y -322.756,Z 932.396,A 0.000,B 0.000,C 90.000,E1 71.329} C_DIS
LIN {X 0.132,Y -312.317,Z 932.384,A 0.000,B 0.000,C 90.000,E1 69.082} C_DIS
LIN {X -0.098,Y -303.429,Z 932.373,A 0.000,B 0.000,C 90.000,E1 67.177} C_DIS
LIN {X 0.018,Y -292.962,Z 932.360,A 0.000,B 0.000,C 90.000,E1 64.845} C_DIS
LIN {X 0.026,Y -282.550,Z 932.347,A 0.000,B 0.000,C 90.000,E1 62.487} C_DIS
LIN {X -0.117,Y -273.519,Z 932.336,A 0.000,B 0.000,C 90.000,E1 60.461} C_DIS
LIN {X -0.037,Y -260.320,Z 932.318,A 0.000,B 0.000,C 90.000,E1 57.296} C_DIS
LIN {X -0.051,Y -248.057,Z 932.300,A 0.000,B 0.000,C 90.000,E1 54.069} C_DIS
LIN {X 0.120,Y -237.030,Z 932.282,A 0.000,B 0.000,C 90.000,E1 50.723} C_DIS
LIN {X -0.023,Y -227.950,Z 932.265,A 0.000,B 0.000,C 90.000,E1 47.757} C_DIS
LIN {X 0.092,Y -219.550,Z 932.248,A 0.000,B 0.000,C 90.000,E1 44.676} C_DIS
LIN {X 0.005,Y -211.794,Z 932.231,A 0.000,B 0.000,C 90.000,E1 41.595} C_DIS
LIN {X -0.073,Y -204.640,Z 932.214,A 0.000,B 0.000,C 90.000,E1 38.463} C_DIS
LIN {X 0.027,Y -197.980,Z 932.196,A 0.000,B 0.000,C 90.000,E1 35.231} C_DIS
LIN {X -0.054,Y -191.823,Z 932.178,A 0.000,B 0.000,C 90.000,E1 32.005} C_DIS
LIN {X 0.007,Y -186.310,Z 932.159,A 0.000,B 0.000,C 90.000,E1 28.693} C_DIS
LIN {X 0.077,Y -181.406,Z 932.141,A 0.000,B 0.000,C 90.000,E1 25.335} C_DIS
LIN {X 0.049,Y -177.224,Z 932.122,A 0.000,B 0.000,C 90.000,E1 21.972} C_DIS
LIN {X 0.107,Y -172.905,Z 932.099,A 0.000,B 0.000,C 90.000,E1 17.692} C_DIS
LIN {X 0.048,Y -169.704,Z 932.075,A 0.000,B 0.000,C 90.000,E1 13.411} C_DIS
LIN {X 0.023,Y -167.265,Z 932.046,A 0.000,B 0.000,C 90.000,E1 8.219} C_DIS
LIN {X -0.042,Y -167.990,Z 931.968,A 0.000,B 0.000,C 90.000,E1 354.318} C_DIS
LIN {X -0.019,Y -171.001,Z 931.939,A 0.000,B 0.000,C 90.000,E1 349.106} C_DIS
LIN {X -0.052,Y -174.630,Z 931.916,A 0.000,B 0.000,C 90.000,E1 344.810} C_DIS
LIN {X -0.082,Y -178.311,Z 931.897,A 0.000,B 0.000,C 90.000,E1 341.402} C_DIS
LIN {X 0.039,Y -182.629,Z 931.878,A 0.000,B 0.000,C 90.000,E1 337.975} C_DIS
LIN {X -0.101,Y -187.712,Z 931.859,A 0.000,B 0.000,C 90.000,E1 334.665} C_DIS
LIN {X 0.041,Y -193.517,Z 931.841,A 0.000,B 0.000,C 90.000,E1 331.307} C_DIS
LIN {X 0.018,Y -200.044,Z 931.823,A 0.000,B 0.000,C 90.000,E1 328.043} C_DIS
LIN {X 0.033,Y -207.058,Z 931.805,A 0.000,B 0.000,C 90.000,E1 324.815} C_DIS
LIN {X -0.045,Y -214.623,Z 931.787,A 0.000,B 0.000,C 90.000,E1 321.662} C_DIS
LIN {X 0.012,Y -222.784,Z 931.770,A 0.000,B 0.000,C 90.000,E1 318.528} C_DIS
LIN {X -0.066,Y -231.792,Z 931.753,A 0.000,B 0.000,C 90.000,E1 315.486} C_DIS
LIN {X 0.081,Y -241.897,Z 931.736,A 0.000,B 0.000,C 90.000,E1 312.447} C_DIS
LIN {X 0.016,Y -251.647,Z 931.722,A 0.000,B 0.000,C 90.000,E1 309.886} C_DIS
LIN {X 0.053,Y -264.235,Z 931.706,A 0.000,B 0.000,C 90.000,E1 306.996} C_DIS
LIN {X -0.029,Y -274.748,Z 931.694,A 0.000,B 0.000,C 90.000,E1 304.898} C_DIS
LIN {X -0.001,Y -291.970,Z 931.677,A 0.000,B 0.000,C 90.000,E1 301.799} C_DIS
LIN {X -0.082,Y -310.797,Z 931.660,A 0.000,B 0.000,C 90.000,E1 298.821} C_DIS
LIN {X 0.034,Y -322.224,Z 931.651,A 0.000,B 0.000,C 90.000,E1 297.180} C_DIS
LIN {X 0.084,Y -339.523,Z 931.639,A 0.000,B 0.000,C 90.000,E1 294.975} C_DIS
LIN {X 0.079,Y -365.260,Z 931.623,A 0.000,B 0.000,C 90.000,E1 292.078} C_DIS
LIN {X -0.136,Y -383.842,Z 931.612,A 0.000,B 0.000,C 90.000,E1 290.174} C_DIS
LIN {X 0.010,Y -399.495,Z 931.603,A 0.000,B 0.000,C 90.000,E1 288.544} C_DIS
LIN {X -0.149,Y -412.299,Z 931.596,A 0.000,B 0.000,C 90.000,E1 287.221} C_DIS
LIN {X -0.122,Y -422.312,Z 931.590,A 0.000,B 0.000,C 90.000,E1 286.134} C_DIS
LIN {X 0.224,Y -431.818,Z 931.584,A 0.000,B 0.000,C 90.000,E1 285.009} C_DIS
LIN {X 0.008,Y -443.002,Z 931.576,A 0.000,B 0.000,C 90.000,E1 283.703} C_DIS
LIN {X 0.041,Y -451.570,Z 931.570,A 0.000,B 0.000,C 90.000,E1 282.647} C_DIS
LIN {X -0.087,Y -461.607,Z 931.563,A 0.000,B 0.000,C 90.000,E1 281.366} C_DIS
LIN {X 0.169,Y -469.029,Z 931.557,A 0.000,B 0.000,C 90.000,E1 280.310} C_DIS
LIN {X 0.101,Y -474.261,Z 931.553,A 0.000,B 0.000,C 90.000,E1 279.557} C_DIS
LIN {X 0.087,Y -478.909,Z 931.549,A 0.000,B 0.000,C 90.000,E1 278.803} C_DIS
LIN {X 0.108,Y -482.887,Z 931.545,A 0.000,B 0.000,C 90.000,E1 278.049} C_DIS
LIN {X -0.200,Y -485.115,Z 931.542,A 0.000,B 0.000,C 90.000,E1 277.587} C_DIS
LIN {X -0.012,Y -487.021,Z 931.539,A 0.000,B 0.000,C 90.000,E1 277.068} C_DIS
LIN {X 0.185,Y -488.616,Z 931.536,A 0.000,B 0.000,C 90.000,E1 276.549} C_DIS
LIN {X -0.094,Y -489.898,Z 931.534,A 0.000,B 0.000,C 90.000,E1 276.087} C_DIS
LIN {X 0.123,Y -490.862,Z 931.531,A 0.000,B 0.000,C 90.000,E1 275.568} C_DIS
LIN {X -0.142,Y -491.465,Z 931.528,A 0.000,B 0.000,C 90.000,E1 275.106} C_DIS
LIN {X 0.084,Y -491.633,Z 931.526,A 0.000,B 0.000,C 90.000,E1 274.588} C_DIS
LIN {X -0.213,Y -491.384,Z 931.523,A 0.000,B 0.000,C 90.000,E1 274.131} C_DIS
LIN {X 0.017,Y -490.644,Z 931.520,A 0.000,B 0.000,C 90.000,E1 273.612} C_DIS
LIN {X 0.240,Y -489.334,Z 931.517,A 0.000,B 0.000,C 90.000,E1 273.094} C_DIS
LIN {X -0.056,Y -487.501,Z 931.515,A 0.000,B 0.000,C 90.000,E1 272.636} C_DIS
LIN {X 0.132,Y -484.941,Z 931.512,A 0.000,B 0.000,C 90.000,E1 272.121} C_DIS
LIN {X -0.165,Y -481.596,Z 931.509,A 0.000,B 0.000,C 90.000,E1 271.661} C_DIS
LIN {X -0.012,Y -477.413,Z 931.506,A 0.000,B 0.000,C 90.000,E1 271.146} C_DIS
LIN {X 0.118,Y -472.200,Z 931.504,A 0.000,B 0.000,C 90.000,E1 270.630} C_DIS
LIN {X 0.043,Y -466.273,Z 931.501,A 0.000,B 0.000,C 90.000,E1 270.172} C_DIS
LIN {X -0.038,Y -460.112,Z 931.499,A 0.000,B 0.000,C 90.000,E1 269.771} C_DIS
LIN {X -0.172,Y -453.506,Z 931.497,A 0.000,B 0.000,C 90.000,E1 269.427} C_DIS
LIN {X 0.149,Y -447.024,Z 931.495,A 0.000,B 0.000,C 90.000,E1 269.083} C_DIS
LIN {X -0.157,Y -440.127,Z 931.494,A 0.000,B 0.000,C 90.000,E1 268.854} C_DIS
LIN {X -0.169,Y -432.876,Z 931.492,A 0.000,B 0.000,C 90.000,E1 268.625} C_DIS
LIN {X 0.120,Y -425.426,Z 931.491,A 0.000,B 0.000,C 90.000,E1 268.396} C_DIS
LIN {X -0.134,Y -416.537,Z 931.490,A 0.000,B 0.000,C 90.000,E1 268.282} C_DIS
LIN {X 0.156,Y -409.558,Z 931.490,A 0.000,B 0.000,C 90.000,E1 268.167} C_DIS
LIN {X -0.007,Y -401.384,Z 931.490,A 0.000,B 0.000,C 90.000,E1 268.165} C_DIS
LIN {X -0.022,Y -181.152,Z 931.490,A 0.000,B 0.000,C 90.000,E1 268.165} C_DIS
LIN {X 0.078,Y -180.786,Z 931.471,A 0.000,B 0.000,C 90.000,E1 264.723} C_DIS
LIN {X -0.027,Y -178.883,Z 931.443,A 0.000,B 0.000,C 90.000,E1 259.690} C_DIS
LIN {X 0.048,Y -175.926,Z 931.414,A 0.000,B 0.000,C 90.000,E1 254.574} C_DIS
LIN {X -0.006,Y -175.365,Z 931.410,A 0.000,B 0.000,C 90.000,E1 253.740} C_DIS
LIN {X 0.052,Y -172.143,Z 931.386,A 0.000,B 0.000,C 90.000,E1 249.444} C_DIS
LIN {X 0.029,Y -171.608,Z 931.381,A 0.000,B 0.000,C 90.000,E1 248.592} C_DIS
LIN {X 0.017,Y -167.831,Z 931.357,A 0.000,B 0.000,C 90.000,E1 244.280} C_DIS
LIN {X 0.035,Y -166.556,Z 931.347,A 0.000,B 0.000,C 90.000,E1 242.538} C_DIS
LIN {X -0.054,Y -162.551,Z 931.323,A 0.000,B 0.000,C 90.000,E1 238.201} C_DIS
LIN {X 0.005,Y -161.229,Z 931.313,A 0.000,B 0.000,C 90.000,E1 236.421} C_DIS
LIN {X 0.040,Y -157.235,Z 931.289,A 0.000,B 0.000,C 90.000,E1 231.984} C_DIS
LIN {X 0.064,Y -155.959,Z 931.279,A 0.000,B 0.000,C 90.000,E1 230.194} C_DIS
LIN {X 0.021,Y -152.213,Z 931.254,A 0.000,B 0.000,C 90.000,E1 225.729} C_DIS
LIN {X 0.042,Y -150.457,Z 931.239,A 0.000,B 0.000,C 90.000,E1 223.014} C_DIS
LIN {X 0.069,Y -147.183,Z 931.214,A 0.000,B 0.000,C 90.000,E1 218.463} C_DIS
LIN {X 0.035,Y -145.201,Z 931.194,A 0.000,B 0.000,C 90.000,E1 214.818} C_DIS
LIN {X -0.055,Y -142.338,Z 931.163,A 0.000,B 0.000,C 90.000,E1 209.333} C_DIS
LIN {X -0.001,Y -141.727,Z 931.153,A 0.000,B 0.000,C 90.000,E1 207.462} C_DIS
LIN {X -0.019,Y -139.480,Z 931.116,A 0.000,B 0.000,C 90.000,E1 200.972} C_DIS
LIN {X -0.030,Y -138.979,Z 931.101,A 0.000,B 0.000,C 90.000,E1 198.181} C_DIS
LIN {X -0.045,Y -138.333,Z 931.054,A 0.000,B 0.000,C 90.000,E1 189.782} C_DIS
LIN {X -0.045,Y -139.429,Z 931.008,A 0.000,B 0.000,C 90.000,E1 181.375} C_DIS
LIN {X 0.008,Y -141.357,Z 930.971,A 0.000,B 0.000,C 90.000,E1 174.837} C_DIS
LIN {X -0.016,Y -142.711,Z 930.956,A 0.000,B 0.000,C 90.000,E1 172.064} C_DIS
LIN {X -0.056,Y -145.086,Z 930.930,A 0.000,B 0.000,C 90.000,E1 167.465} C_DIS
LIN {X -0.061,Y -147.710,Z 930.910,A 0.000,B 0.000,C 90.000,E1 163.795} C_DIS
LIN {X 0.022,Y -150.365,Z 930.890,A 0.000,B 0.000,C 90.000,E1 160.115} C_DIS
LIN {X 0.041,Y -153.792,Z 930.869,A 0.000,B 0.000,C 90.000,E1 156.485} C_DIS
LIN {X -0.039,Y -157.204,Z 930.849,A 0.000,B 0.000,C 90.000,E1 152.922} C_DIS
LIN {X 0.042,Y -161.366,Z 930.830,A 0.000,B 0.000,C 90.000,E1 149.331} C_DIS
LIN {X 0.053,Y -165.569,Z 930.810,A 0.000,B 0.000,C 90.000,E1 145.801} C_DIS
LIN {X -0.063,Y -170.486,Z 930.791,A 0.000,B 0.000,C 90.000,E1 142.351} C_DIS
LIN {X 0.086,Y -175.368,Z 930.772,A 0.000,B 0.000,C 90.000,E1 138.852} C_DIS
LIN {X -0.052,Y -180.992,Z 930.753,A 0.000,B 0.000,C 90.000,E1 135.486} C_DIS
LIN {X 0.073,Y -186.419,Z 930.734,A 0.000,B 0.000,C 90.000,E1 132.081} C_DIS
LIN {X -0.126,Y -191.046,Z 930.720,A 0.000,B 0.000,C 90.000,E1 129.644} C_DIS
LIN {X 0.010,Y -194.072,Z 930.710,A 0.000,B 0.000,C 90.000,E1 127.810} C_DIS
LIN {X -0.020,Y -296.657,Z 930.710,A 0.000,B 0.000,C 90.000,E1 127.810} C_DIS
LIN {X 0.125,Y -299.017,Z 930.710,A 0.000,B 0.000,C 90.000,E1 127.729} C_DIS
LIN {X 0.006,Y -304.162,Z 930.708,A 0.000,B 0.000,C 90.000,E1 127.443} C_DIS
LIN {X -0.116,Y -307.026,Z 930.706,A 0.000,B 0.000,C 90.000,E1 127.156} C_DIS
LIN {X -0.187,Y -309.052,Z 930.705,A 0.000,B 0.000,C 90.000,E1 126.870} C_DIS
LIN {X -0.008,Y -310.638,Z 930.703,A 0.000,B 0.000,C 90.000,E1 126.537} C_DIS
LIN {X -0.035,Y -312.004,Z 930.701,A 0.000,B 0.000,C 90.000,E1 126.217} C_DIS
LIN {X 0.062,Y -324.556,Z 930.680,A 0.000,B 0.000,C 90.000,E1 122.339} C_DIS
LIN {X -0.152,Y -335.369,Z 930.664,A 0.000,B 0.000,C 90.000,E1 119.539} C_DIS
LIN {X -0.089,Y -347.557,Z 930.648,A 0.000,B 0.000,C 90.000,E1 116.744} C_DIS
LIN {X 0.003,Y -361.237,Z 930.633,A 0.000,B 0.000,C 90.000,E1 114.003} C_DIS
LIN {X -0.060,Y -374.742,Z 930.620,A 0.000,B 0.000,C 90.000,E1 111.642} C_DIS
LIN {X -0.059,Y -389.614,Z 930.607,A 0.000,B 0.000,C 90.000,E1 109.322} C_DIS
LIN {X 0.071,Y -405.959,Z 930.595,A 0.000,B 0.000,C 90.000,E1 107.040} C_DIS
LIN {X 0.104,Y -423.896,Z 930.582,A 0.000,B 0.000,C 90.000,E1 104.828} C_DIS
LIN {X 0.037,Y -443.424,Z 930.571,A 0.000,B 0.000,C 90.000,E1 102.703} C_DIS
LIN {X 0.150,Y -463.707,Z 930.560,A 0.000,B 0.000,C 90.000,E1 100.715} C_DIS
LIN {X 0.097,Y -468.561,Z 930.557,A 0.000,B 0.000,C 90.000,E1 100.254} C_DIS
LIN {X -0.026,Y -470.396,Z 930.556,A 0.000,B 0.000,C 90.000,E1 100.018} C_DIS
LIN {X -0.150,Y -471.779,Z 930.554,A 0.000,B 0.000,C 90.000,E1 99.782} C_DIS
LIN {X -0.053,Y -473.560,Z 930.551,A 0.000,B 0.000,C 90.000,E1 99.265} C_DIS
LIN {X 0.057,Y -474.254,Z 930.549,A 0.000,B 0.000,C 90.000,E1 98.746} C_DIS
LIN {X 0.248,Y -473.981,Z 930.546,A 0.000,B 0.000,C 90.000,E1 98.219} C_DIS
LIN {X -0.096,Y -472.705,Z 930.543,A 0.000,B 0.000,C 90.000,E1 97.757} C_DIS
LIN {X 0.168,Y -471.629,Z 930.542,A 0.000,B 0.000,C 90.000,E1 97.473} C_DIS
LIN {X -0.120,Y -468.533,Z 930.539,A 0.000,B 0.000,C 90.000,E1 97.004} C_DIS
LIN {X 0.150,Y -452.470,Z 930.525,A 0.000,B 0.000,C 90.000,E1 94.416} C_DIS
LIN {X -0.178,Y -441.266,Z 930.515,A 0.000,B 0.000,C 90.000,E1 92.636} C_DIS
LIN {X 0.121,Y -429.892,Z 930.504,A 0.000,B 0.000,C 90.000,E1 90.745} C_DIS
LIN {X 0.079,Y -414.067,Z 930.489,A 0.000,B 0.000,C 90.000,E1 88.051} C_DIS
LIN {X -0.173,Y -403.151,Z 930.479,A 0.000,B 0.000,C 90.000,E1 86.159} C_DIS
LIN {X -0.200,Y -392.216,Z 930.468,A 0.000,B 0.000,C 90.000,E1 84.204} C_DIS
LIN {X -0.024,Y -381.194,Z 930.457,A 0.000,B 0.000,C 90.000,E1 82.186} C_DIS
LIN {X 0.019,Y -371.593,Z 930.447,A 0.000,B 0.000,C 90.000,E1 80.443} C_DIS
LIN {X -0.110,Y -361.703,Z 930.437,A 0.000,B 0.000,C 90.000,E1 78.701} C_DIS
LIN {X 0.073,Y -351.667,Z 930.427,A 0.000,B 0.000,C 90.000,E1 76.881} C_DIS
LIN {X 0.058,Y -338.366,Z 930.414,A 0.000,B 0.000,C 90.000,E1 74.448} C_DIS
LIN {X -0.102,Y -321.277,Z 930.395,A 0.000,B 0.000,C 90.000,E1 71.040} C_DIS
LIN {X -0.029,Y -309.403,Z 930.380,A 0.000,B 0.000,C 90.000,E1 68.465} C_DIS
LIN {X 0.087,Y -300.463,Z 930.369,A 0.000,B 0.000,C 90.000,E1 66.485} C_DIS
LIN {X -0.119,Y -291.534,Z 930.358,A 0.000,B 0.000,C 90.000,E1 64.537} C_DIS
LIN {X -0.008,Y -281.095,Z 930.345,A 0.000,B 0.000,C 90.000,E1 62.153} C_DIS
LIN {X 0.063,Y -272.057,Z 930.334,A 0.000,B 0.000,C 90.000,E1 60.078} C_DIS
LIN {X -0.038,Y -260.329,Z 930.318,A 0.000,B 0.000,C 90.000,E1 57.296} C_DIS
LIN {X -0.053,Y -248.063,Z 930.300,A 0.000,B 0.000,C 90.000,E1 54.069} C_DIS
LIN {X 0.119,Y -237.066,Z 930.282,A 0.000,B 0.000,C 90.000,E1 50.723} C_DIS
LIN {X -0.024,Y -228.018,Z 930.265,A 0.000,B 0.000,C 90.000,E1 47.757} C_DIS
LIN {X 0.094,Y -219.647,Z 930.248,A 0.000,B 0.000,C 90.000,E1 44.676} C_DIS
LIN {X 0.010,Y -211.920,Z 930.231,A 0.000,B 0.000,C 90.000,E1 41.595} C_DIS
LIN {X -0.065,Y -204.798,Z 930.214,A 0.000,B 0.000,C 90.000,E1 38.463} C_DIS
LIN {X 0.038,Y -198.161,Z 930.196,A 0.000,B 0.000,C 90.000,E1 35.231} C_DIS
LIN {X -0.039,Y -192.030,Z 930.178,A 0.000,B 0.000,C 90.000,E1 32.005} C_DIS
LIN {X 0.026,Y -186.520,Z 930.159,A 0.000,B 0.000,C 90.000,E1 28.693} C_DIS
LIN {X 0.102,Y -181.604,Z 930.141,A 0.000,B 0.000,C 90.000,E1 25.335} C_DIS
LIN {X -0.087,Y -177.417,Z 930.122,A 0.000,B 0.000,C 90.000,E1 22.025} C_DIS
LIN {X -0.077,Y -173.110,Z 930.099,A 0.000,B 0.000,C 90.000,E1 17.764} C_DIS
LIN {X 0.087,Y -169.925,Z 930.075,A 0.000,B 0.000,C 90.000,E1 13.411} C_DIS
LIN {X 0.070,Y -167.492,Z 930.046,A 0.000,B 0.000,C 90.000,E1 8.219} C_DIS
LIN {X -0.033,Y -168.254,Z 929.968,A 0.000,B 0.000,C 90.000,E1 354.318} C_DIS
LIN {X -0.035,Y -170.660,Z 929.944,A 0.000,B 0.000,C 90.000,E1 349.982} C_DIS
LIN {X 0.049,Y -174.070,Z 929.920,A 0.000,B 0.000,C 90.000,E1 345.644} C_DIS
LIN {X 0.007,Y -177.565,Z 929.901,A 0.000,B 0.000,C 90.000,E1 342.236} C_DIS
LIN {X -0.010,Y -181.741,Z 929.882,A 0.000,B 0.000,C 90.000,E1 338.847} C_DIS
LIN {X -0.006,Y -186.611,Z 929.864,A 0.000,B 0.000,C 90.000,E1 335.485} C_DIS
LIN {X 0.024,Y -192.260,Z 929.845,A 0.000,B 0.000,C 90.000,E1 332.153} C_DIS
LIN {X 0.038,Y -198.627,Z 929.827,A 0.000,B 0.000,C 90.000,E1 328.869} C_DIS
LIN {X -0.101,Y -205.531,Z 929.809,A 0.000,B 0.000,C 90.000,E1 325.674} C_DIS
LIN {X -0.057,Y -212.968,Z 929.791,A 0.000,B 0.000,C 90.000,E1 322.477} C_DIS
LIN {X 0.117,Y -220.937,Z 929.774,A 0.000,B 0.000,C 90.000,E1 319.299} C_DIS
LIN {X -0.004,Y -229.722,Z 929.757,A 0.000,B 0.000,C 90.000,E1 316.257} C_DIS
LIN {X 0.090,Y -239.504,Z 929.740,A 0.000,B 0.000,C 90.000,E1 313.218} C_DIS
LIN {X -0.058,Y -250.415,Z 929.724,A 0.000,B 0.000,C 90.000,E1 310.297} C_DIS
LIN {X 0.101,Y -261.153,Z 929.710,A 0.000,B 0.000,C 90.000,E1 307.729} C_DIS
LIN {X 0.122,Y -271.234,Z 929.698,A 0.000,B 0.000,C 90.000,E1 305.598} C_DIS
LIN {X 0.058,Y -288.073,Z 929.681,A 0.000,B 0.000,C 90.000,E1 302.498} C_DIS
LIN {X 0.027,Y -306.422,Z 929.664,A 0.000,B 0.000,C 90.000,E1 299.489} C_DIS
LIN {X 0.079,Y -317.424,Z 929.655,A 0.000,B 0.000,C 90.000,E1 297.847} C_DIS
LIN {X -0.076,Y -334.302,Z 929.642,A 0.000,B 0.000,C 90.000,E1 295.643} C_DIS
LIN {X -0.041,Y -357.757,Z 929.627,A 0.000,B 0.000,C 90.000,E1 292.898} C_DIS
LIN {X -0.081,Y -376.411,Z 929.616,A 0.000,B 0.000,C 90.000,E1 290.918} C_DIS
LIN {X 0.025,Y -392.187,Z 929.607,A 0.000,B 0.000,C 90.000,E1 289.268} C_DIS
LIN {X -0.113,Y -405.184,Z 929.600,A 0.000,B 0.000,C 90.000,E1 287.946} C_DIS
LIN {X -0.053,Y -415.363,Z 929.594,A 0.000,B 0.000,C 90.000,E1 286.858} C_DIS
LIN {X -0.062,Y -425.184,Z 929.588,A 0.000,B 0.000,C 90.000,E1 285.788} C_DIS
LIN {X 0.116,Y -432.222,Z 929.583,A 0.000,B 0.000,C 90.000,E1 284.954} C_DIS
LIN {X -0.094,Y -443.438,Z 929.576,A 0.000,B 0.000,C 90.000,E1 283.647} C_DIS
LIN {X -0.056,Y -451.986,Z 929.570,A 0.000,B 0.000,C 90.000,E1 282.591} C_DIS
LIN {X -0.087,Y -461.973,Z 929.563,A 0.000,B 0.000,C 90.000,E1 281.299} C_DIS
LIN {X 0.083,Y -469.385,Z 929.557,A 0.000,B 0.000,C 90.000,E1 280.254} C_DIS
LIN {X 0.019,Y -474.608,Z 929.553,A 0.000,B 0.000,C 90.000,E1 279.500} C_DIS
LIN {X 0.007,Y -479.217,Z 929.549,A 0.000,B 0.000,C 90.000,E1 278.746} C_DIS
LIN {X 0.225,Y -481.952,Z 929.546,A 0.000,B 0.000,C 90.000,E1 278.219} C_DIS
LIN {X 0.206,Y -485.363,Z 929.542,A 0.000,B 0.000,C 90.000,E1 277.473} C_DIS
LIN {X -0.026,Y -487.255,Z 929.539,A 0.000,B 0.000,C 90.000,E1 277.004} C_DIS
LIN {X 0.169,Y -488.849,Z 929.536,A 0.000,B 0.000,C 90.000,E1 276.486} C_DIS
LIN {X -0.112,Y -490.079,Z 929.533,A 0.000,B 0.000,C 90.000,E1 276.024} C_DIS
LIN {X 0.055,Y -490.993,Z 929.531,A 0.000,B 0.000,C 90.000,E1 275.511} C_DIS
LIN {X -0.210,Y -491.547,Z 929.528,A 0.000,B 0.000,C 90.000,E1 275.049} C_DIS
LIN {X 0.018,Y -491.669,Z 929.525,A 0.000,B 0.000,C 90.000,E1 274.531} C_DIS
LIN {X 0.246,Y -491.387,Z 929.522,A 0.000,B 0.000,C 90.000,E1 274.012} C_DIS
LIN {X -0.048,Y -490.560,Z 929.520,A 0.000,B 0.000,C 90.000,E1 273.555} C_DIS
LIN {X 0.176,Y -489.201,Z 929.517,A 0.000,B 0.000,C 90.000,E1 273.037} C_DIS
LIN {X -0.120,Y -487.287,Z 929.514,A 0.000,B 0.000,C 90.000,E1 272.579} C_DIS
LIN {X 0.068,Y -484.668,Z 929.512,A 0.000,B 0.000,C 90.000,E1 272.064} C_DIS
LIN {X -0.230,Y -481.283,Z 929.509,A 0.000,B 0.000,C 90.000,E1 271.604} C_DIS
LIN {X -0.078,Y -476.985,Z 929.506,A 0.000,B 0.000,C 90.000,E1 271.088} C_DIS
LIN {X 0.052,Y -471.661,Z 929.503,A 0.000,B 0.000,C 90.000,E1 270.573} C_DIS
LIN {X 0.030,Y -465.751,Z 929.501,A 0.000,B 0.000,C 90.000,E1 270.115} C_DIS
LIN {X -0.010,Y -459.587,Z 929.498,A 0.000,B 0.000,C 90.000,E1 269.714} C_DIS
LIN {X -0.136,Y -452.922,Z 929.496,A 0.000,B 0.000,C 90.000,E1 269.370} C_DIS
LIN {X 0.187,Y -446.281,Z 929.495,A 0.000,B 0.000,C 90.000,E1 269.026} C_DIS
LIN {X -0.114,Y -439.214,Z 929.493,A 0.000,B 0.000,C 90.000,E1 268.797} C_DIS
LIN {X -0.058,Y -432.166,Z 929.492,A 0.000,B 0.000,C 90.000,E1 268.568} C_DIS
LIN {X -0.165,Y -424.626,Z 929.491,A 0.000,B 0.000,C 90.000,E1 268.396} C_DIS
LIN {X 0.044,Y -415.611,Z 929.490,A 0.000,B 0.000,C 90.000,E1 268.224} C_DIS
LIN {X -0.039,Y -407.693,Z 929.490,A 0.000,B 0.000,C 90.000,E1 268.165} C_DIS
LIN {X -0.128,Y -403.668,Z 929.490,A 0.000,B 0.000,C 90.000,E1 268.165} C_DIS
LIN {X -0.078,Y -181.148,Z 929.490,A 0.000,B 0.000,C 90.000,E1 268.165} C_DIS
LIN {X -0.087,Y -180.902,Z 929.474,A 0.000,B 0.000,C 90.000,E1 265.298} C_DIS
LIN {X 0.043,Y -180.230,Z 929.464,A 0.000,B 0.000,C 90.000,E1 263.571} C_DIS
LIN {X 0.059,Y -178.714,Z 929.441,A 0.000,B 0.000,C 90.000,E1 259.342} C_DIS
LIN {X -0.048,Y -175.763,Z 929.413,A 0.000,B 0.000,C 90.000,E1 254.283} C_DIS
LIN {X 0.002,Y -171.946,Z 929.384,A 0.000,B 0.000,C 90.000,E1 249.135} C_DIS
LIN {X -0.023,Y -171.332,Z 929.379,A 0.000,B 0.000,C 90.000,E1 248.284} C_DIS
LIN {X 0.030,Y -167.587,Z 929.355,A 0.000,B 0.000,C 90.000,E1 243.948} C_DIS
LIN {X -0.031,Y -166.224,Z 929.346,A 0.000,B 0.000,C 90.000,E1 242.231} C_DIS
LIN {X -0.042,Y -162.986,Z 929.326,A 0.000,B 0.000,C 90.000,E1 238.742} C_DIS
LIN {X 0.005,Y -160.903,Z 929.312,A 0.000,B 0.000,C 90.000,E1 236.087} C_DIS
LIN {X -0.018,Y -157.669,Z 929.292,A 0.000,B 0.000,C 90.000,E1 232.557} C_DIS
LIN {X -0.079,Y -155.707,Z 929.277,A 0.000,B 0.000,C 90.000,E1 229.908} C_DIS
LIN {X -0.024,Y -151.969,Z 929.252,A 0.000,B 0.000,C 90.000,E1 225.405} C_DIS
LIN {X -0.008,Y -150.211,Z 929.237,A 0.000,B 0.000,C 90.000,E1 222.690} C_DIS
LIN {X -0.084,Y -146.977,Z 929.212,A 0.000,B 0.000,C 90.000,E1 218.177} C_DIS
LIN {X 0.026,Y -145.564,Z 929.197,A 0.000,B 0.000,C 90.000,E1 215.391} C_DIS
LIN {X 0.025,Y -142.955,Z 929.171,A 0.000,B 0.000,C 90.000,E1 210.797} C_DIS
LIN {X -0.045,Y -141.581,Z 929.151,A 0.000,B 0.000,C 90.000,E1 207.129} C_DIS
LIN {X 0.003,Y -139.417,Z 929.115,A 0.000,B 0.000,C 90.000,E1 200.610} C_DIS
LIN {X 0.055,Y -139.141,Z 929.104,A 0.000,B 0.000,C 90.000,E1 198.725} C_DIS
LIN {X -0.054,Y -138.347,Z 929.057,A 0.000,B 0.000,C 90.000,E1 190.366} C_DIS
LIN {X 0.070,Y -139.491,Z 929.006,A 0.000,B 0.000,C 90.000,E1 180.974} C_DIS
LIN {X 0.011,Y -141.101,Z 928.975,A 0.000,B 0.000,C 90.000,E1 175.412} C_DIS
LIN {X -0.036,Y -142.480,Z 928.959,A 0.000,B 0.000,C 90.000,E1 172.648} C_DIS
LIN {X 0.054,Y -144.729,Z 928.933,A 0.000,B 0.000,C 90.000,E1 167.993} C_DIS
LIN {X 0.004,Y -147.333,Z 928.913,A 0.000,B 0.000,C 90.000,E1 164.338} C_DIS
LIN {X 0.069,Y -150.656,Z 928.888,A 0.000,B 0.000,C 90.000,E1 159.752} C_DIS
LIN {X -0.050,Y -154.135,Z 928.868,A 0.000,B 0.000,C 90.000,E1 156.177} C_DIS
LIN {X 0.013,Y -157.562,Z 928.848,A 0.000,B 0.000,C 90.000,E1 152.564} C_DIS
LIN {X 0.038,Y -161.805,Z 928.828,A 0.000,B 0.000,C 90.000,E1 148.997} C_DIS
LIN {X 0.057,Y -165.997,Z 928.808,A 0.000,B 0.000,C 90.000,E1 145.468} C_DIS
LIN {X 0.050,Y -170.995,Z 928.789,A 0.000,B 0.000,C 90.000,E1 141.984} C_DIS
LIN {X -0.035,Y -175.864,Z 928.770,A 0.000,B 0.000,C 90.000,E1 138.566} C_DIS
LIN {X -0.041,Y -181.470,Z 928.751,A 0.000,B 0.000,C 90.000,E1 135.162} C_DIS
LIN {X 0.096,Y -186.981,Z 928.732,A 0.000,B 0.000,C 90.000,E1 131.757} C_DIS
LIN {X 0.098,Y -190.097,Z 928.723,A 0.000,B 0.000,C 90.000,E1 130.092} C_DIS
LIN {X -0.037,Y -194.018,Z 928.710,A 0.000,B 0.000,C 90.000,E1 127.855} C_DIS
LIN {X 0.142,Y -296.413,Z 928.710,A 0.000,B 0.000,C 90.000,E1 127.810} C_DIS
LIN {X -0.023,Y -301.791,Z 928.709,A 0.000,B 0.000,C 90.000,E1 127.649} C_DIS
LIN {X 0.030,Y -304.807,Z 928.708,A 0.000,B 0.000,C 90.000,E1 127.397} C_DIS
LIN {X -0.101,Y -308.536,Z 928.705,A 0.000,B 0.000,C 90.000,E1 126.950} C_DIS
LIN {X 0.109,Y -310.346,Z 928.703,A 0.000,B 0.000,C 90.000,E1 126.583} C_DIS
LIN {X -0.118,Y -311.760,Z 928.702,A 0.000,B 0.000,C 90.000,E1 126.297} C_DIS
LIN {X 0.006,Y -315.804,Z 928.694,A 0.000,B 0.000,C 90.000,E1 124.978} C_DIS
LIN {X -0.116,Y -326.593,Z 928.677,A 0.000,B 0.000,C 90.000,E1 121.799} C_DIS
LIN {X 0.019,Y -337.669,Z 928.661,A 0.000,B 0.000,C 90.000,E1 118.949} C_DIS
LIN {X -0.007,Y -350.149,Z 928.645,A 0.000,B 0.000,C 90.000,E1 116.181} C_DIS
LIN {X 0.026,Y -364.136,Z 928.630,A 0.000,B 0.000,C 90.000,E1 113.462} C_DIS
LIN {X 0.049,Y -377.939,Z 928.617,A 0.000,B 0.000,C 90.000,E1 111.099} C_DIS
LIN {X 0.141,Y -393.133,Z 928.604,A 0.000,B 0.000,C 90.000,E1 108.779} C_DIS
LIN {X -0.023,Y -409.825,Z 928.592,A 0.000,B 0.000,C 90.000,E1 106.551} C_DIS
LIN {X -0.016,Y -428.137,Z 928.580,A 0.000,B 0.000,C 90.000,E1 104.356} C_DIS
LIN {X 0.048,Y -447.904,Z 928.568,A 0.000,B 0.000,C 90.000,E1 102.243} C_DIS
LIN {X 0.019,Y -468.130,Z 928.557,A 0.000,B 0.000,C 90.000,E1 100.310} C_DIS
LIN {X 0.049,Y -469.944,Z 928.556,A 0.000,B 0.000,C 90.000,E1 100.074} C_DIS
LIN {X -0.182,Y -471.453,Z 928.555,A 0.000,B 0.000,C 90.000,E1 99.849} C_DIS
LIN {X 0.134,Y -472.581,Z 928.553,A 0.000,B 0.000,C 90.000,E1 99.557} C_DIS
LIN {X -0.152,Y -473.927,Z 928.550,A 0.000,B 0.000,C 90.000,E1 99.086} C_DIS
LIN {X -0.039,Y -474.256,Z 928.548,A 0.000,B 0.000,C 90.000,E1 98.568} C_DIS
LIN {X 0.084,Y -473.622,Z 928.545,A 0.000,B 0.000,C 90.000,E1 98.049} C_DIS
LIN {X 0.210,Y -471.926,Z 928.542,A 0.000,B 0.000,C 90.000,E1 97.530} C_DIS
LIN {X 0.069,Y -470.586,Z 928.541,A 0.000,B 0.000,C 90.000,E1 97.296} C_DIS
LIN {X -0.016,Y -454.489,Z 928.526,A 0.000,B 0.000,C 90.000,E1 94.759} C_DIS
LIN {X -0.082,Y -444.974,Z 928.518,A 0.000,B 0.000,C 90.000,E1 93.212} C_DIS
LIN {X -0.118,Y -433.663,Z 928.508,A 0.000,B 0.000,C 90.000,E1 91.375} C_DIS
LIN {X -0.169,Y -419.180,Z 928.494,A 0.000,B 0.000,C 90.000,E1 88.969} C_DIS
LIN {X 0.093,Y -408.280,Z 928.484,A 0.000,B 0.000,C 90.000,E1 87.020} C_DIS
LIN {X -0.194,Y -395.764,Z 928.471,A 0.000,B 0.000,C 90.000,E1 84.837} C_DIS
LIN {X 0.056,Y -384.784,Z 928.460,A 0.000,B 0.000,C 90.000,E1 82.818} C_DIS
LIN {X 0.107,Y -375.258,Z 928.451,A 0.000,B 0.000,C 90.000,E1 81.084} C_DIS
LIN {X 0.041,Y -365.480,Z 928.441,A 0.000,B 0.000,C 90.000,E1 79.342} C_DIS
LIN {X -0.098,Y -353.807,Z 928.429,A 0.000,B 0.000,C 90.000,E1 77.285} C_DIS
LIN {X -0.140,Y -342.107,Z 928.417,A 0.000,B 0.000,C 90.000,E1 75.172} C_DIS
LIN {X -0.172,Y -324.730,Z 928.398,A 0.000,B 0.000,C 90.000,E1 71.764} C_DIS
LIN {X -0.122,Y -312.765,Z 928.384,A 0.000,B 0.000,C 90.000,E1 69.209} C_DIS
LIN {X 0.058,Y -303.885,Z 928.374,A 0.000,B 0.000,C 90.000,E1 67.230} C_DIS
LIN {X 0.055,Y -293.458,Z 928.361,A 0.000,B 0.000,C 90.000,E1 64.921} C_DIS
LIN {X 0.071,Y -283.023,Z 928.348,A 0.000,B 0.000,C 90.000,E1 62.564} C_DIS
LIN {X -0.127,Y -272.491,Z 928.334,A 0.000,B 0.000,C 90.000,E1 60.205} C_DIS
LIN {X 0.012,Y -260.721,Z 928.319,A 0.000,B 0.000,C 90.000,E1 57.375} C_DIS
LIN {X 0.007,Y -248.414,Z 928.301,A 0.000,B 0.000,C 90.000,E1 54.149} C_DIS
LIN {X -0.006,Y -237.413,Z 928.282,A 0.000,B 0.000,C 90.000,E1 50.848} C_DIS
LIN {X -0.007,Y -227.315,Z 928.264,A 0.000,B 0.000,C 90.000,E1 47.472} C_DIS
LIN {X -0.062,Y -219.045,Z 928.247,A 0.000,B 0.000,C 90.000,E1 44.433} C_DIS
LIN {X 0.002,Y -211.369,Z 928.229,A 0.000,B 0.000,C 90.000,E1 41.310} C_DIS
LIN {X -0.083,Y -204.328,Z 928.212,A 0.000,B 0.000,C 90.000,E1 38.177} C_DIS
LIN {X 0.009,Y -197.770,Z 928.194,A 0.000,B 0.000,C 90.000,E1 34.945} C_DIS
LIN {X 0.083,Y -191.700,Z 928.176,A 0.000,B 0.000,C 90.000,E1 31.671} C_DIS
LIN {X -0.027,Y -186.249,Z 928.158,A 0.000,B 0.000,C 90.000,E1 28.409} C_DIS
LIN {X -0.044,Y -181.410,Z 928.139,A 0.000,B 0.000,C 90.000,E1 25.079} C_DIS
LIN {X -0.071,Y -177.255,Z 928.121,A 0.000,B 0.000,C 90.000,E1 21.716} C_DIS
LIN {X -0.068,Y -173.042,Z 928.097,A 0.000,B 0.000,C 90.000,E1 17.457} C_DIS
LIN {X 0.047,Y -169.950,Z 928.073,A 0.000,B 0.000,C 90.000,E1 13.119} C_DIS
LIN {X 0.004,Y -167.397,Z 928.039,A 0.000,B 0.000,C 90.000,E1 7.068} C_DIS
LIN {X -0.023,Y -168.529,Z 927.968,A 0.000,B 0.000,C 90.000,E1 354.318} C_DIS
LIN {X -0.017,Y -170.930,Z 927.944,A 0.000,B 0.000,C 90.000,E1 349.982} C_DIS
LIN {X 0.076,Y -174.344,Z 927.920,A 0.000,B 0.000,C 90.000,E1 345.644} C_DIS
LIN {X 0.042,Y -177.824,Z 927.901,A 0.000,B 0.000,C 90.000,E1 342.236} C_DIS
LIN {X 0.031,Y -181.994,Z 927.883,A 0.000,B 0.000,C 90.000,E1 338.847} C_DIS
LIN {X 0.043,Y -186.856,Z 927.864,A 0.000,B 0.000,C 90.000,E1 335.485} C_DIS
LIN {X 0.081,Y -192.520,Z 927.845,A 0.000,B 0.000,C 90.000,E1 332.153} C_DIS
LIN {X 0.103,Y -198.905,Z 927.827,A 0.000,B 0.000,C 90.000,E1 328.869} C_DIS
LIN {X -0.026,Y -205.818,Z 927.809,A 0.000,B 0.000,C 90.000,E1 325.674} C_DIS
LIN {X 0.028,Y -213.251,Z 927.792,A 0.000,B 0.000,C 90.000,E1 322.477} C_DIS
LIN {X -0.032,Y -222.257,Z 927.772,A 0.000,B 0.000,C 90.000,E1 318.976} C_DIS
LIN {X 0.044,Y -231.141,Z 927.755,A 0.000,B 0.000,C 90.000,E1 315.891} C_DIS
LIN {X 0.004,Y -241.046,Z 927.738,A 0.000,B 0.000,C 90.000,E1 312.894} C_DIS
LIN {X 0.071,Y -250.645,Z 927.724,A 0.000,B 0.000,C 90.000,E1 310.297} C_DIS
LIN {X -0.125,Y -261.342,Z 927.710,A 0.000,B 0.000,C 90.000,E1 307.810} C_DIS
LIN {X 0.050,Y -271.375,Z 927.698,A 0.000,B 0.000,C 90.000,E1 305.644} C_DIS
LIN {X -0.025,Y -288.098,Z 927.681,A 0.000,B 0.000,C 90.000,E1 302.546} C_DIS
LIN {X -0.070,Y -306.369,Z 927.664,A 0.000,B 0.000,C 90.000,E1 299.539} C_DIS
LIN {X -0.025,Y -317.312,Z 927.655,A 0.000,B 0.000,C 90.000,E1 297.897} C_DIS
LIN {X 0.017,Y -334.034,Z 927.643,A 0.000,B 0.000,C 90.000,E1 295.668} C_DIS
LIN {X 0.112,Y -356.968,Z 927.628,A 0.000,B 0.000,C 90.000,E1 292.950} C_DIS
LIN {X 0.063,Y -375.555,Z 927.617,A 0.000,B 0.000,C 90.000,E1 290.972} C_DIS
LIN {X 0.069,Y -391.395,Z 927.607,A 0.000,B 0.000,C 90.000,E1 289.322} C_DIS
LIN {X -0.043,Y -404.342,Z 927.600,A 0.000,B 0.000,C 90.000,E1 288.000} C_DIS
LIN {X 0.026,Y -414.568,Z 927.594,A 0.000,B 0.000,C 90.000,E1 286.913} C_DIS
LIN {X -0.096,Y -424.543,Z 927.588,A 0.000,B 0.000,C 90.000,E1 285.843} C_DIS
LIN {X 0.091,Y -431.614,Z 927.583,A 0.000,B 0.000,C 90.000,E1 285.009} C_DIS
LIN {X -0.131,Y -442.891,Z 927.576,A 0.000,B 0.000,C 90.000,E1 283.703} C_DIS
LIN {X -0.102,Y -451.459,Z 927.570,A 0.000,B 0.000,C 90.000,E1 282.647} C_DIS
LIN {X -0.236,Y -461.478,Z 927.563,A 0.000,B 0.000,C 90.000,E1 281.366} C_DIS
LIN {X 0.017,Y -468.935,Z 927.557,A 0.000,B 0.000,C 90.000,E1 280.310} C_DIS
LIN {X -0.053,Y -474.191,Z 927.553,A 0.000,B 0.000,C 90.000,E1 279.557} C_DIS
LIN {X -0.071,Y -478.872,Z 927.549,A 0.000,B 0.000,C 90.000,E1 278.803} C_DIS
LIN {X -0.051,Y -482.901,Z 927.545,A 0.000,B 0.000,C 90.000,E1 278.049} C_DIS
LIN {X 0.123,Y -485.146,Z 927.542,A 0.000,B 0.000,C 90.000,E1 277.530} C_DIS
LIN {X -0.171,Y -487.104,Z 927.539,A 0.000,B 0.000,C 90.000,E1 277.068} C_DIS
LIN {X 0.025,Y -488.721,Z 927.536,A 0.000,B 0.000,C 90.000,E1 276.549} C_DIS
LIN {X -0.254,Y -490.005,Z 927.534,A 0.000,B 0.000,C 90.000,E1 276.087} C_DIS
LIN {X -0.036,Y -490.954,Z 927.531,A 0.000,B 0.000,C 90.000,E1 275.568} C_DIS
LIN {X 0.188,Y -491.552,Z 927.528,A 0.000,B 0.000,C 90.000,E1 275.049} C_DIS
LIN {X -0.075,Y -491.736,Z 927.525,A 0.000,B 0.000,C 90.000,E1 274.588} C_DIS
LIN {X 0.118,Y -491.497,Z 927.523,A 0.000,B 0.000,C 90.000,E1 274.073} C_DIS
LIN {X -0.141,Y -490.763,Z 927.520,A 0.000,B 0.000,C 90.000,E1 273.612} C_DIS
LIN {X 0.084,Y -489.467,Z 927.517,A 0.000,B 0.000,C 90.000,E1 273.094} C_DIS
LIN {X -0.211,Y -487.625,Z 927.515,A 0.000,B 0.000,C 90.000,E1 272.636} C_DIS
LIN {X -0.022,Y -485.106,Z 927.512,A 0.000,B 0.000,C 90.000,E1 272.121} C_DIS
LIN {X 0.164,Y -481.821,Z 927.509,A 0.000,B 0.000,C 90.000,E1 271.604} C_DIS
LIN {X -0.162,Y -477.629,Z 927.506,A 0.000,B 0.000,C 90.000,E1 271.146} C_DIS
LIN {X -0.028,Y -472.453,Z 927.503,A 0.000,B 0.000,C 90.000,E1 270.630} C_DIS
LIN {X -0.143,Y -466.596,Z 927.501,A 0.000,B 0.000,C 90.000,E1 270.172} C_DIS
LIN {X 0.164,Y -460.319,Z 927.499,A 0.000,B 0.000,C 90.000,E1 269.714} C_DIS
LIN {X -0.026,Y -453.614,Z 927.496,A 0.000,B 0.000,C 90.000,E1 269.370} C_DIS
LIN {X -0.192,Y -447.011,Z 927.495,A 0.000,B 0.000,C 90.000,E1 269.083} C_DIS
LIN {X -0.076,Y -440.009,Z 927.493,A 0.000,B 0.000,C 90.000,E1 268.797} C_DIS
LIN {X -0.076,Y -432.855,Z 927.492,A 0.000,B 0.000,C 90.000,E1 268.568} C_DIS
LIN {X -0.215,Y -425.482,Z 927.491,A 0.000,B 0.000,C 90.000,E1 268.396} C_DIS
LIN {X -0.082,Y -415.900,Z 927.490,A 0.000,B 0.000,C 90.000,E1 268.224} C_DIS
LIN {X -0.162,Y -408.131,Z 927.490,A 0.000,B 0.000,C 90.000,E1 268.165} C_DIS
LIN {X 0.156,Y -404.963,Z 927.490,A 0.000,B 0.000,C 90.000,E1 268.108} C_DIS
LIN {X 0.050,Y -181.145,Z 927.490,A 0.000,B 0.000,C 90.000,E1 268.108} C_DIS
LIN {X 0.040,Y -180.900,Z 927.474,A 0.000,B 0.000,C 90.000,E1 265.241} C_DIS
LIN {X -0.010,Y -180.223,Z 927.464,A 0.000,B 0.000,C 90.000,E1 263.571} C_DIS
LIN {X -0.057,Y -179.038,Z 927.445,A 0.000,B 0.000,C 90.000,E1 260.208} C_DIS
LIN {X 0.006,Y -178.703,Z 927.441,A 0.000,B 0.000,C 90.000,E1 259.342} C_DIS
LIN {X -0.053,Y -175.753,Z 927.412,A 0.000,B 0.000,C 90.000,E1 254.267} C_DIS
LIN {X -0.050,Y -171.936,Z 927.384,A 0.000,B 0.000,C 90.000,E1 249.135} C_DIS
LIN {X -0.074,Y -171.316,Z 927.379,A 0.000,B 0.000,C 90.000,E1 248.284} C_DIS
LIN {X -0.021,Y -167.575,Z 927.355,A 0.000,B 0.000,C 90.000,E1 243.948} C_DIS
LIN {X -0.082,Y -166.206,Z 927.346,A 0.000,B 0.000,C 90.000,E1 242.231} C_DIS
LIN {X -0.092,Y -162.972,Z 927.326,A 0.000,B 0.000,C 90.000,E1 238.742} C_DIS
LIN {X -0.045,Y -160.884,Z 927.312,A 0.000,B 0.000,C 90.000,E1 236.087} C_DIS
LIN {X -0.067,Y -157.655,Z 927.292,A 0.000,B 0.000,C 90.000,E1 232.557} C_DIS
LIN {X 0.092,Y -155.692,Z 927.277,A 0.000,B 0.000,C 90.000,E1 229.828} C_DIS
LIN {X -0.072,Y -151.956,Z 927.252,A 0.000,B 0.000,C 90.000,E1 225.405} C_DIS
LIN {X -0.055,Y -150.196,Z 927.237,A 0.000,B 0.000,C 90.000,E1 222.690} C_DIS
LIN {X 0.075,Y -146.967,Z 927.212,A 0.000,B 0.000,C 90.000,E1 218.096} C_DIS
LIN {X -0.021,Y -145.554,Z 927.197,A 0.000,B 0.000,C 90.000,E1 215.391} C_DIS
LIN {X -0.021,Y -142.947,Z 927.171,A 0.000,B 0.000,C 90.000,E1 210.797} C_DIS
LIN {X 0.035,Y -141.572,Z 927.151,A 0.000,B 0.000,C 90.000,E1 207.078} C_DIS
LIN {X -0.043,Y -139.413,Z 927.114,A 0.000,B 0.000,C 90.000,E1 200.610} C_DIS
LIN {X 0.009,Y -139.136,Z 927.104,A 0.000,B 0.000,C 90.000,E1 198.725} C_DIS
LIN {X 0.037,Y -138.349,Z 927.057,A 0.000,B 0.000,C 90.000,E1 190.310} C_DIS
LIN {X 0.024,Y -139.495,Z 927.005,A 0.000,B 0.000,C 90.000,E1 180.974} C_DIS
LIN {X -0.035,Y -141.110,Z 926.974,A 0.000,B 0.000,C 90.000,E1 175.412} C_DIS
LIN {X 0.059,Y -142.489,Z 926.959,A 0.000,B 0.000,C 90.000,E1 172.591} C_DIS
LIN {X 0.007,Y -144.741,Z 926.933,A 0.000,B 0.000,C 90.000,E1 167.993} C_DIS
LIN {X -0.043,Y -147.348,Z 926.913,A 0.000,B 0.000,C 90.000,E1 164.338} C_DIS
LIN {X 0.021,Y -150.672,Z 926.888,A 0.000,B 0.000,C 90.000,E1 159.752} C_DIS
LIN {X -0.098,Y -154.151,Z 926.867,A 0.000,B 0.000,C 90.000,E1 156.177} C_DIS
LIN {X 0.037,Y -157.581,Z 926.848,A 0.000,B 0.000,C 90.000,E1 152.538} C_DIS
LIN {X -0.013,Y -161.828,Z 926.828,A 0.000,B 0.000,C 90.000,E1 148.997} C_DIS
LIN {X 0.006,Y -166.020,Z 926.808,A 0.000,B 0.000,C 90.000,E1 145.468} C_DIS
LIN {X -0.002,Y -171.020,Z 926.789,A 0.000,B 0.000,C 90.000,E1 141.984} C_DIS
LIN {X 0.029,Y -175.891,Z 926.770,A 0.000,B 0.000,C 90.000,E1 138.528} C_DIS
